// TwinCAT 3 PLC project PLC
// ProgramVersion: 3.1.4026.19
// libraries:
//   Tc2_Standard, * (Beckhoff Automation GmbH)
//   Tc2_System, * (Beckhoff Automation GmbH)
//   Tc2_Utilities, * (Beckhoff Automation GmbH)
//   Tc3_IotBase, * (Beckhoff Automation GmbH)
//   Tc3_IotCommunicator, * (Beckhoff Automation GmbH)
// project tree:
//   DUTs/10-IoT/ ST_IoT_Communicator.TcDUT
//   GVLs/01-System/ GVL_ADS.TcGVL, GVL_NovRam.TcGVL, GVL_System.TcGVL
//   GVLs/02-Knoppen/ GVL_Deurcontacten.TcGVL, GVL_Drukknoppen.TcGVL
//   GVLs/03-Verlichting/ GVL_Dimmers.TcGVL, GVL_Relais.TcGVL
//   GVLs/04-Boiler/ GVL_Boiler.TcGVL
//   GVLs/05-Temperaturen/ GVL_Temperaturen.TcGVL
//   GVLs/06-Screens/ GVL_Screens.TcGVL
//   GVLs/07-Draaipoort/ GVL_Draaipoort.TcGVL
//   GVLs/08-Energiemetingen/ GVL_Energiemetingen.TcGVL
//   GVLs/09-Ventilatie/ GVL_Ventilatie.TcGVL
//   GVLs/90-Visualisatie/ GVL_Visualisatie.TcGVL
//   / PlcTask.TcTTO
//   POUs/00-MAIN/ MAIN.TcPOU
//   POUs/01-System/ P_SunriseSunset.TcPOU, P_WinTime.TcPOU
//   POUs/02-Knoppen/ P_Doors.TcPOU, P_Drukknoppen.TcPOU
//   POUs/03-Verlichting/ P_LightsBerging.TcPOU, P_LightsBoven.TcPOU, P_LightsBuiten.TcPOU, P_LightsHal.TcPOU, P_LightsKeukenLiving.TcPOU, P_LightsLeefruimte.TcPOU
//   POUs/04-Boiler/ P_Boiler.TcPOU
//   POUs/05-Temperaturen/ P_Temperatures.TcPOU
//   POUs/06-Screens/ P_Screens.TcPOU
//   POUs/07-Draaipoort/ P_Draaipoort.TcPOU
//   POUs/08-Energiemetingen/ P_Kwartierpiek.TcPOU, P_Watermeting.TcPOU
//   POUs/09-Ventilatie/ P_Ventilatie.TcPOU
//   POUs/10-IoT/ P_IoT_Communicator.TcPOU, P_Sonos.TcPOU (not stored)
//   POUs/99-FB%27s/ FB_Dimmer.TcPOU (not stored), FB_LongMultipleClick.TcPOU (not stored), FB_OnOffLight.TcPOU (not stored), FB_Screens.TcPOU (not stored)
// real-time tasks:
//   TASK PlcTask: cycle T#10ms, priority 20, ADS port 350
// I/O:
//   DEVICE Device 1 (NOV-DP-RAM)
//     Box 2 (Retain Handler)
//   DEVICE Device 2 (Onboard I/O Device), AmsNetId 5.170.212.74.3.1
//     Term 1 (CX7028) [CX7028-0000-0121]
//       modules: Module 1 (DIO_2x), Module 2 (Empty Module), Module 3 (DIO_2x), Module 4 (Empty Module), Module 5 (DI_2x), Module 6 (Empty Module), Module 7 (DI_2x), Module 8 (Empty Module)
//   DEVICE Device 3 (EtherCAT), AmsNetId 192.168.0.199.4.1
//     Term 1 (EK1200) [EK1200-7000 EtherCAT Power supply (1,5A E-Bus)]
//       DK01-02-03-04 (EL1809) [EL1809 16Ch. Dig. Input 24V, 3ms]
//       DK04-05-06-07 (EL1809) [EL1809 16Ch. Dig. Input 24V, 3ms]
//       DK08-11-12 (EL1809) [EL1809 16Ch. Dig. Input 24V, 3ms]
//       DK13-14-15-16 (EL1809) [EL1809 16Ch. Dig. Input 24V, 3ms]
//       DK09-10 (EL1809) [EL1809 16Ch. Dig. Input 24V, 3ms]
//       Sensoren (EL1008) [EL1008 8Ch. Dig. Input 24V, 3ms]
//       Lights J-K (EL2809) [EL2809 16Ch. Dig. Output 24V, 0.5A]
//       Lights X-Y (EL2809) [EL2809 16Ch. Dig. Output 24V, 0.5A]
//       Boiler en poort (EL2809) [EL2809 16Ch. Dig. Output 24V, 0.5A]
//       Temperaturen (EL3208) [EL3208 8Ch. Ana. Input PT100 (RTD)]
//       Ventilatie en Dimmers1 (EL4004) [EL4004 4Ch. Ana. Output 0-10V, 12bit]
//       Term 15 (EL6851) [EL6851 DMX Master]
//       Term 16 (EL3403) [EL3403 3Ch. Power Measuring]
//       Term 17 (EK1122) [EK1122 2 port EtherCAT junction]
//         Kast Tuinhuis (EK1828) [EK1828 EtherCAT IO-Coupler  (1A E-Bus, 4 Ch. Dig. In, 3ms, 8 Ch. Dig. Out 24V, 0,5A)]
//         Kast Tuinhuis achteraan (EK1828) [EK1828 EtherCAT IO-Coupler  (1A E-Bus, 4 Ch. Dig. In, 3ms, 8 Ch. Dig. Out 24V, 0,5A)]
//         Kast Verdieping (EK1100) [EK1100 EtherCAT Coupler (2A E-Bus)]
//           DK17-18-19 (EL1809) [EL1809 16Ch. Dig. Input 24V, 3ms]
//           DK20-21-22 (EL1809) [EL1809 16Ch. Dig. Input 24V, 3ms]
//           Term 23 (EL1809) [EL1809 16Ch. Dig. Input 24V, 3ms]
//           Screens en Lights-BD (EL2809) [EL2809 16Ch. Dig. Output 24V, 0.5A]
//           Rolluiken (EL2008) [EL2008 8Ch. Dig. Output 24V, 0.5A]
//           Dimmers2 (EL4008) [EL4008 8Ch. Ana. Output 0-10V, 12bit]
//           Term 27 (EL3064) [EL3064 4Ch. Ana. Input 0-10V]
//           Term 26 (EL9011) [EL9011 End Terminal]
// variable links:
//   (this object) <-> Device 1 (NOV-DP-RAM)/Box 2 (Retain Handler)
//     PlcTask Retains/GVL_NovRam.bNovRamBoiler <-> Retains/GVL_NovRam.bNovRamBoiler_[851]
//     PlcTask Retains/GVL_NovRam.bNovRamLight_BD{2..8} <-> Retains/GVL_NovRam.bNovRamLight_BD{2..8}_[851]  (7 links)
//     PlcTask Retains/GVL_NovRam.bNovRamLight_I{1..8} <-> Retains/GVL_NovRam.bNovRamLight_I{1..8}_[851]  (8 links)
//     PlcTask Retains/GVL_NovRam.bNovRamLight_J{3..6} <-> Retains/GVL_NovRam.bNovRamLight_J{3..6}_[851]  (4 links)
//     PlcTask Retains/GVL_NovRam.bNovRamLight_W{1..8} <-> Retains/GVL_NovRam.bNovRamLight_W{1..8}_[851]  (8 links)
//     PlcTask Retains/GVL_NovRam.bNovRamLight_Y{1..7} <-> Retains/GVL_NovRam.bNovRamLight_Y{1..7}_[851]  (7 links)
//     PlcTask Retains/GVL_NovRam.bNovRamLight_Z{1..4} <-> Retains/GVL_NovRam.bNovRamLight_Z{1..4}_[851]  (4 links)
//     PlcTask Retains/GVL_NovRam.bNovRamLight_ZZ{1..6} <-> Retains/GVL_NovRam.bNovRamLight_ZZ{1..6}_[851]  (6 links)
//     PlcTask Retains/GVL_NovRam.diWaterteller <-> Retains/GVL_NovRam.diWaterteller_[851]
//     PlcTask Retains/GVL_NovRam.diWatertellerGisteren <-> Retains/GVL_NovRam.diWatertellerGisteren_[851]
//     PlcTask Retains/GVL_NovRam.iNovRamVentilatie <-> Retains/GVL_NovRam.iNovRamVentilatie_[851]
//     PlcTask Retains/GVL_NovRam.nDimmValue_BD1 <-> Retains/GVL_NovRam.nDimmValue_BD1_[851]
//     PlcTask Retains/GVL_NovRam.nDimmValue_I2 <-> Retains/GVL_NovRam.nDimmValue_I2_[851]
//     PlcTask Retains/GVL_NovRam.nDimmValue_J1 <-> Retains/GVL_NovRam.nDimmValue_J1_[851]
//     PlcTask Retains/GVL_NovRam.nDimmValue_J2 <-> Retains/GVL_NovRam.nDimmValue_J2_[851]
//   (this object) <-> Device 3 (EtherCAT)/Term 1 (EK1200)/Boiler en poort (EL2809)
//     PlcTask Outputs/GVL_Boiler.bRelaisBoiler <-> Channel 1/GVL_Boiler.bRelaisBoiler
//     PlcTask Outputs/GVL_Draaipoort.bDraaipoortVoetgangerOpenDicht <-> Channel 3/GVL_Draaipoort.bDraaipoortVoetgangerOpenDicht
//     PlcTask Outputs/GVL_Draaipoort.bDraaipoortVolledigOpenDicht <-> Channel 2/GVL_Draaipoort.bDraaipoortVolledigOpenDicht
//   (this object) <-> Device 3 (EtherCAT)/Term 1 (EK1200)/DK01-02-03-04 (EL1809)
//     PlcTask Inputs/GVL_Drukknoppen.bDK01x1 <-> Channel 1/GVL_Drukknoppen.bDK01x1
//     PlcTask Inputs/GVL_Drukknoppen.bDK01x2 <-> Channel 2/GVL_Drukknoppen.bDK01x2
//     PlcTask Inputs/GVL_Drukknoppen.bDK01x3 <-> Channel 3/GVL_Drukknoppen.bDK01x3
//     PlcTask Inputs/GVL_Drukknoppen.bDK01x4 <-> Channel 4/GVL_Drukknoppen.bDK01x4
//     PlcTask Inputs/GVL_Drukknoppen.bDK01x5 <-> Channel 5/GVL_Drukknoppen.bDK01x5
//     PlcTask Inputs/GVL_Drukknoppen.bDK01x6 <-> Channel 6/GVL_Drukknoppen.bDK01x6
//     PlcTask Inputs/GVL_Drukknoppen.bDK02x1 <-> Channel 7/GVL_Drukknoppen.bDK02x1
//     PlcTask Inputs/GVL_Drukknoppen.bDK03x1 <-> Channel 9/GVL_Drukknoppen.bDK03x1
//     PlcTask Inputs/GVL_Drukknoppen.bDK03x2 <-> Channel 10/GVL_Drukknoppen.bDK03x2
//     PlcTask Inputs/GVL_Drukknoppen.bDK03x3 <-> Channel 11/GVL_Drukknoppen.bDK03x3
//     PlcTask Inputs/GVL_Drukknoppen.bDK03x4 <-> Channel 12/GVL_Drukknoppen.bDK03x4
//     PlcTask Inputs/GVL_Drukknoppen.bDK04x1 <-> Channel 13/GVL_Drukknoppen.bDK04x1
//     PlcTask Inputs/GVL_Drukknoppen.bDK04x2 <-> Channel 14/GVL_Drukknoppen.bDK04x2
//     PlcTask Inputs/GVL_Drukknoppen.bDK04x3 <-> Channel 15/GVL_Drukknoppen.bDK04x3
//     PlcTask Inputs/GVL_Drukknoppen.bDK04x4 <-> Channel 16/GVL_Drukknoppen.bDK04x4
//   (this object) <-> Device 3 (EtherCAT)/Term 1 (EK1200)/DK04-05-06-07 (EL1809)
//     PlcTask Inputs/GVL_Drukknoppen.bDK04x5 <-> Channel 1/GVL_Drukknoppen.bDK04x5
//     PlcTask Inputs/GVL_Drukknoppen.bDK04x6 <-> Channel 2/GVL_Drukknoppen.bDK04x6
//     PlcTask Inputs/GVL_Drukknoppen.bDK05x1 <-> Channel 3/GVL_Drukknoppen.bDK05x1
//     PlcTask Inputs/GVL_Drukknoppen.bDK05x2 <-> Channel 4/GVL_Drukknoppen.bDK05x2
//     PlcTask Inputs/GVL_Drukknoppen.bDK05x3 <-> Channel 5/GVL_Drukknoppen.bDK05x3
//     PlcTask Inputs/GVL_Drukknoppen.bDK05x4 <-> Channel 6/GVL_Drukknoppen.bDK05x4
//     PlcTask Inputs/GVL_Drukknoppen.bDK06x1 <-> Channel 7/GVL_Drukknoppen.bDK06x1
//     PlcTask Inputs/GVL_Drukknoppen.bDK06x2 <-> Channel 8/GVL_Drukknoppen.bDK06x2
//     PlcTask Inputs/GVL_Drukknoppen.bDK06x3 <-> Channel 9/GVL_Drukknoppen.bDK06x3
//     PlcTask Inputs/GVL_Drukknoppen.bDK06x4 <-> Channel 10/GVL_Drukknoppen.bDK06x4
//     PlcTask Inputs/GVL_Drukknoppen.bDK07x1 <-> Channel 11/GVL_Drukknoppen.bDK07x1
//     PlcTask Inputs/GVL_Drukknoppen.bDK07x2 <-> Channel 12/GVL_Drukknoppen.bDK07x2
//     PlcTask Inputs/GVL_Drukknoppen.bDK07x3 <-> Channel 13/GVL_Drukknoppen.bDK07x3
//     PlcTask Inputs/GVL_Drukknoppen.bDK07x4 <-> Channel 14/GVL_Drukknoppen.bDK07x4
//     PlcTask Inputs/GVL_Drukknoppen.bDK07x5 <-> Channel 15/GVL_Drukknoppen.bDK07x5
//     PlcTask Inputs/GVL_Drukknoppen.bDK07x6 <-> Channel 16/GVL_Drukknoppen.bDK07x6
//   (this object) <-> Device 3 (EtherCAT)/Term 1 (EK1200)/DK08-11-12 (EL1809)
//     PlcTask Inputs/GVL_Drukknoppen.bDK08x1 <-> Channel 1/GVL_Drukknoppen.bDK08x1
//     PlcTask Inputs/GVL_Drukknoppen.bDK08x2 <-> Channel 2/GVL_Drukknoppen.bDK08x2
//     PlcTask Inputs/GVL_Drukknoppen.bDK08x3 <-> Channel 3/GVL_Drukknoppen.bDK08x3
//     PlcTask Inputs/GVL_Drukknoppen.bDK08x4 <-> Channel 4/GVL_Drukknoppen.bDK08x4
//     PlcTask Inputs/GVL_Drukknoppen.bDK11x1 <-> Channel 9/GVL_Drukknoppen.bDK11x1
//     PlcTask Inputs/GVL_Drukknoppen.bDK11x2 <-> Channel 10/GVL_Drukknoppen.bDK11x2
//     PlcTask Inputs/GVL_Drukknoppen.bDK11x3 <-> Channel 11/GVL_Drukknoppen.bDK11x3
//     PlcTask Inputs/GVL_Drukknoppen.bDK11x4 <-> Channel 12/GVL_Drukknoppen.bDK11x4
//     PlcTask Inputs/GVL_Drukknoppen.bDK12x1 <-> Channel 13/GVL_Drukknoppen.bDK12x1
//     PlcTask Inputs/GVL_Drukknoppen.bDK12x2 <-> Channel 14/GVL_Drukknoppen.bDK12x2
//     PlcTask Inputs/GVL_Drukknoppen.bDK12x3 <-> Channel 15/GVL_Drukknoppen.bDK12x3
//     PlcTask Inputs/GVL_Drukknoppen.bDK12x4 <-> Channel 16/GVL_Drukknoppen.bDK12x4
//   (this object) <-> Device 3 (EtherCAT)/Term 1 (EK1200)/DK09-10 (EL1809)
//     PlcTask Inputs/GVL_Drukknoppen.bDK09x1 <-> Channel 1/GVL_Drukknoppen.bDK09x1
//     PlcTask Inputs/GVL_Drukknoppen.bDK09x2 <-> Channel 2/GVL_Drukknoppen.bDK09x2
//     PlcTask Inputs/GVL_Drukknoppen.bDK09x3 <-> Channel 3/GVL_Drukknoppen.bDK09x3
//     PlcTask Inputs/GVL_Drukknoppen.bDK09x4 <-> Channel 4/GVL_Drukknoppen.bDK09x4
//     PlcTask Inputs/GVL_Drukknoppen.bDK09x5 <-> Channel 5/GVL_Drukknoppen.bDK09x5
//     PlcTask Inputs/GVL_Drukknoppen.bDK09x6 <-> Channel 6/GVL_Drukknoppen.bDK09x6
//     PlcTask Inputs/GVL_Drukknoppen.bDK10x1 <-> Channel 7/GVL_Drukknoppen.bDK10x1
//     PlcTask Inputs/GVL_Drukknoppen.bDK10x2 <-> Channel 8/GVL_Drukknoppen.bDK10x2
//     PlcTask Inputs/GVL_Drukknoppen.bDK10x3 <-> Channel 9/GVL_Drukknoppen.bDK10x3
//     PlcTask Inputs/GVL_Drukknoppen.bDK10x4 <-> Channel 10/GVL_Drukknoppen.bDK10x4
//     PlcTask Inputs/GVL_Drukknoppen.bDK10x5 <-> Channel 11/GVL_Drukknoppen.bDK10x5
//     PlcTask Inputs/GVL_Drukknoppen.bDK10x6 <-> Channel 12/GVL_Drukknoppen.bDK10x6
//   (this object) <-> Device 3 (EtherCAT)/Term 1 (EK1200)/DK13-14-15-16 (EL1809)
//     PlcTask Inputs/GVL_Drukknoppen.bDK13x1 <-> Channel 1/GVL_Drukknoppen.bDK13x1
//     PlcTask Inputs/GVL_Drukknoppen.bDK13x2 <-> Channel 2/GVL_Drukknoppen.bDK13x2
//     PlcTask Inputs/GVL_Drukknoppen.bDK13x3 <-> Channel 3/GVL_Drukknoppen.bDK13x3
//     PlcTask Inputs/GVL_Drukknoppen.bDK13x4 <-> Channel 4/GVL_Drukknoppen.bDK13x4
//     PlcTask Inputs/GVL_Drukknoppen.bDK14x1 <-> Channel 5/GVL_Drukknoppen.bDK14x1
//     PlcTask Inputs/GVL_Drukknoppen.bDK14x2 <-> Channel 6/GVL_Drukknoppen.bDK14x2
//     PlcTask Inputs/GVL_Drukknoppen.bDK14x3 <-> Channel 7/GVL_Drukknoppen.bDK14x3
//     PlcTask Inputs/GVL_Drukknoppen.bDK14x4 <-> Channel 8/GVL_Drukknoppen.bDK14x4
//     PlcTask Inputs/GVL_Drukknoppen.bDK15x1 <-> Channel 9/GVL_Drukknoppen.bDK15x1
//     PlcTask Inputs/GVL_Drukknoppen.bDK15x2 <-> Channel 10/GVL_Drukknoppen.bDK15x2
//     PlcTask Inputs/GVL_Drukknoppen.bDK15x3 <-> Channel 11/GVL_Drukknoppen.bDK15x3
//     PlcTask Inputs/GVL_Drukknoppen.bDK15x4 <-> Channel 12/GVL_Drukknoppen.bDK15x4
//     PlcTask Inputs/GVL_Drukknoppen.bDK16x1 <-> Channel 13/GVL_Drukknoppen.bDK16x1
//     PlcTask Inputs/GVL_Drukknoppen.bDK16x2 <-> Channel 14/GVL_Drukknoppen.bDK16x2
//     PlcTask Inputs/GVL_Drukknoppen.bDK16x3 <-> Channel 15/GVL_Drukknoppen.bDK16x3
//     PlcTask Inputs/GVL_Drukknoppen.bDK16x4 <-> Channel 16/GVL_Drukknoppen.bDK16x4
//   (this object) <-> Device 3 (EtherCAT)/Term 1 (EK1200)/Lights J-K (EL2809)
//     PlcTask Outputs/GVL_Drukknoppen.bMeldingDK02x1 <-> Channel 15/GVL_Drukknoppen.bMeldingDK02x1
//     PlcTask Outputs/GVL_Drukknoppen.bMeldingDK11x3 <-> Channel 16/GVL_Drukknoppen.bMeldingDK11x3
//     PlcTask Outputs/GVL_Relais.bRelaisLight_I{1..8} <-> Channel {1..8}/GVL_Relais.bRelaisLight_I{1..8}  (8 links)
//     PlcTask Outputs/GVL_Relais.bRelaisLight_J1 <-> Channel 9/GVL_Relais.bRelaisLight_J1
//     PlcTask Outputs/GVL_Relais.bRelaisLight_J3 <-> Channel 11/GVL_Relais.bRelaisLight_J3
//     PlcTask Outputs/GVL_Relais.bRelaisLight_J4 <-> Channel 12/GVL_Relais.bRelaisLight_J4
//     PlcTask Outputs/GVL_Relais.bRelaisLight_J5 <-> Channel 13/GVL_Relais.bRelaisLight_J5
//     PlcTask Outputs/GVL_Relais.bRelaisLight_J6 <-> Channel 14/GVL_Relais.bRelaisLight_J6
//   (this object) <-> Device 3 (EtherCAT)/Term 1 (EK1200)/Lights X-Y (EL2809)
//     PlcTask Outputs/GVL_Drukknoppen.bMeldingDK11x4 <-> Channel 16/GVL_Drukknoppen.bMeldingDK11x4
//     PlcTask Outputs/GVL_Relais.bRelaisLight_W{1..8} <-> Channel {1..8}/GVL_Relais.bRelaisLight_W{1..8}  (8 links)
//     PlcTask Outputs/GVL_Relais.bRelaisLight_Y{1..7} <-> Channel {9..15}/GVL_Relais.bRelaisLight_Y{1..7}  (7 links)
//   (this object) <-> Device 3 (EtherCAT)/Term 1 (EK1200)/Sensoren (EL1008)
//     PlcTask Inputs/GVL_Deurcontacten.bContactSchuifdeur <-> Channel 3/GVL_Deurcontacten.bContactSchuifdeur
//     PlcTask Inputs/GVL_Deurcontacten.bContactSchuifdeurLeefruimte <-> Channel 4/GVL_Deurcontacten.bContactSchuifdeurLeefruimte
//     PlcTask Inputs/GVL_Deurcontacten.bContactVoordeur <-> Channel 1/GVL_Deurcontacten.bContactVoordeur
//     PlcTask Inputs/GVL_Deurcontacten.bContactZijdeur <-> Channel 2/GVL_Deurcontacten.bContactZijdeur
//     PlcTask Inputs/GVL_Energiemetingen.bWaterSensor <-> Channel 7/GVL_Energiemetingen.bWaterSensor
//   (this object) <-> Device 3 (EtherCAT)/Term 1 (EK1200)/Temperaturen (EL3208)
//     PlcTask Inputs/GVL_Temperaturen.iTemp{1..8} <-> RTD Inputs Channel {1..8}/GVL_Temperaturen.iTemp{1..8}  (8 links)
//   (this object) <-> Device 3 (EtherCAT)/Term 1 (EK1200)/Term 17 (EK1122)/Kast Tuinhuis (EK1828)
//     PlcTask Inputs/GVL_Drukknoppen.bDK30x1 <-> Channel 1/GVL_Drukknoppen.bDK30x1
//     PlcTask Inputs/GVL_Drukknoppen.bDK30x2 <-> Channel 2/GVL_Drukknoppen.bDK30x2
//     PlcTask Outputs/GVL_Relais.bRelaisLight_Z{1..4} <-> Channel {5..8}/GVL_Relais.bRelaisLight_Z{1..4}  (4 links)
//   (this object) <-> Device 3 (EtherCAT)/Term 1 (EK1200)/Term 17 (EK1122)/Kast Tuinhuis achteraan (EK1828)
//     PlcTask Inputs/GVL_Drukknoppen.bDK40x{1..4} <-> Channel {1..4}/GVL_Drukknoppen.bDK40x{1..4}  (4 links)
//     PlcTask Outputs/GVL_Relais.bRelaisLight_ZZ{1..6} <-> Channel {5..10}/GVL_Relais.bRelaisLight_ZZ{1..6}  (6 links)
//   (this object) <-> Device 3 (EtherCAT)/Term 1 (EK1200)/Term 17 (EK1122)/Kast Verdieping (EK1100)/DK17-18-19 (EL1809)
//     PlcTask Inputs/GVL_Drukknoppen.bDK17x1 <-> Channel 1/GVL_Drukknoppen.bDK17x1
//     PlcTask Inputs/GVL_Drukknoppen.bDK17x2 <-> Channel 2/GVL_Drukknoppen.bDK17x2
//     PlcTask Inputs/GVL_Drukknoppen.bDK17x3 <-> Channel 3/GVL_Drukknoppen.bDK17x3
//     PlcTask Inputs/GVL_Drukknoppen.bDK17x4 <-> Channel 4/GVL_Drukknoppen.bDK17x4
//     PlcTask Inputs/GVL_Drukknoppen.bDK17x5 <-> Channel 5/GVL_Drukknoppen.bDK17x5
//     PlcTask Inputs/GVL_Drukknoppen.bDK17x6 <-> Channel 6/GVL_Drukknoppen.bDK17x6
//     PlcTask Inputs/GVL_Drukknoppen.bDK18x1 <-> Channel 7/GVL_Drukknoppen.bDK18x1
//     PlcTask Inputs/GVL_Drukknoppen.bDK18x2 <-> Channel 8/GVL_Drukknoppen.bDK18x2
//     PlcTask Inputs/GVL_Drukknoppen.bDK18x3 <-> Channel 9/GVL_Drukknoppen.bDK18x3
//     PlcTask Inputs/GVL_Drukknoppen.bDK18x4 <-> Channel 10/GVL_Drukknoppen.bDK18x4
//     PlcTask Inputs/GVL_Drukknoppen.bDK19x1 <-> Channel 11/GVL_Drukknoppen.bDK19x1
//     PlcTask Inputs/GVL_Drukknoppen.bDK19x2 <-> Channel 12/GVL_Drukknoppen.bDK19x2
//     PlcTask Inputs/GVL_Drukknoppen.bDK19x3 <-> Channel 13/GVL_Drukknoppen.bDK19x3
//     PlcTask Inputs/GVL_Drukknoppen.bDK19x4 <-> Channel 14/GVL_Drukknoppen.bDK19x4
//     PlcTask Inputs/GVL_Drukknoppen.bDK19x5 <-> Channel 15/GVL_Drukknoppen.bDK19x5
//     PlcTask Inputs/GVL_Drukknoppen.bDK19x6 <-> Channel 16/GVL_Drukknoppen.bDK19x6
//   (this object) <-> Device 3 (EtherCAT)/Term 1 (EK1200)/Term 17 (EK1122)/Kast Verdieping (EK1100)/DK20-21-22 (EL1809)
//     PlcTask Inputs/GVL_Drukknoppen.bDK20x1 <-> Channel 1/GVL_Drukknoppen.bDK20x1
//     PlcTask Inputs/GVL_Drukknoppen.bDK20x2 <-> Channel 2/GVL_Drukknoppen.bDK20x2
//     PlcTask Inputs/GVL_Drukknoppen.bDK20x3 <-> Channel 3/GVL_Drukknoppen.bDK20x3
//     PlcTask Inputs/GVL_Drukknoppen.bDK20x4 <-> Channel 4/GVL_Drukknoppen.bDK20x4
//     PlcTask Inputs/GVL_Drukknoppen.bDK21x1 <-> Channel 5/GVL_Drukknoppen.bDK21x1
//     PlcTask Inputs/GVL_Drukknoppen.bDK21x2 <-> Channel 6/GVL_Drukknoppen.bDK21x2
//     PlcTask Inputs/GVL_Drukknoppen.bDK21x3 <-> Channel 7/GVL_Drukknoppen.bDK21x3
//     PlcTask Inputs/GVL_Drukknoppen.bDK21x4 <-> Channel 8/GVL_Drukknoppen.bDK21x4
//     PlcTask Inputs/GVL_Drukknoppen.bDK22x1 <-> Channel 9/GVL_Drukknoppen.bDK22x1
//     PlcTask Inputs/GVL_Drukknoppen.bDK22x2 <-> Channel 10/GVL_Drukknoppen.bDK22x2
//     PlcTask Inputs/GVL_Drukknoppen.bDK22x3 <-> Channel 11/GVL_Drukknoppen.bDK22x3
//     PlcTask Inputs/GVL_Drukknoppen.bDK22x4 <-> Channel 12/GVL_Drukknoppen.bDK22x4
//   (this object) <-> Device 3 (EtherCAT)/Term 1 (EK1200)/Term 17 (EK1122)/Kast Verdieping (EK1100)/Dimmers2 (EL4008)
//     PlcTask Outputs/GVL_Dimmers.DimLight_BD1 <-> AO Outputs Channel 1/GVL_Dimmers.DimLight_BD1
//   (this object) <-> Device 3 (EtherCAT)/Term 1 (EK1200)/Term 17 (EK1122)/Kast Verdieping (EK1100)/Rolluiken (EL2008)
//     PlcTask Outputs/GVL_Screens.bMotorRolluik2Omhoog <-> Channel 1/GVL_Screens.bMotorRolluik2Omhoog
//     PlcTask Outputs/GVL_Screens.bMotorRolluik3Omhoog <-> Channel 3/GVL_Screens.bMotorRolluik3Omhoog
//     PlcTask Outputs/GVL_Screens.bMotorRolluik2Omlaag <-> Channel 2/GVL_Screens.bMotorRolluik2Omlaag
//     PlcTask Outputs/GVL_Screens.bMotorRolluik3Omlaag <-> Channel 4/GVL_Screens.bMotorRolluik3Omlaag
//   (this object) <-> Device 3 (EtherCAT)/Term 1 (EK1200)/Term 17 (EK1122)/Kast Verdieping (EK1100)/Screens en Lights-BD (EL2809)
//     PlcTask Outputs/GVL_Relais.bRelaisLight_BD2 <-> Channel 11/GVL_Relais.bRelaisLight_BD2
//     PlcTask Outputs/GVL_Relais.bRelaisLight_BD3 <-> Channel 12/GVL_Relais.bRelaisLight_BD3
//     PlcTask Outputs/GVL_Relais.bRelaisLight_BD4 <-> Channel 13/GVL_Relais.bRelaisLight_BD4
//     PlcTask Outputs/GVL_Relais.bRelaisLight_BD5 <-> Channel 14/GVL_Relais.bRelaisLight_BD5
//     PlcTask Outputs/GVL_Relais.bRelaisLight_BD6 <-> Channel 15/GVL_Relais.bRelaisLight_BD6
//     PlcTask Outputs/GVL_Relais.bRelaisLight_BD8 <-> Channel 16/GVL_Relais.bRelaisLight_BD8
//     PlcTask Outputs/GVL_Screens.bMotorRolluik1Omhoog <-> Channel 9/GVL_Screens.bMotorRolluik1Omhoog
//     PlcTask Outputs/GVL_Screens.bMotorRolluik1Omlaag <-> Channel 10/GVL_Screens.bMotorRolluik1Omlaag
//     PlcTask Outputs/GVL_Screens.bMotorScreen{1..4}Omhoog <-> Channel {1..7 step 2}/GVL_Screens.bMotorScreen{1..4}Omhoog  (4 links)
//     PlcTask Outputs/GVL_Screens.bMotorScreen{1..4}Omlaag <-> Channel {2..8 step 2}/GVL_Screens.bMotorScreen{1..4}Omlaag  (4 links)
//   (this object) <-> Device 3 (EtherCAT)/Term 1 (EK1200)/Ventilatie en Dimmers1 (EL4004)
//     PlcTask Outputs/GVL_Dimmers.DimLight_I2 <-> AO Outputs Channel 2/GVL_Dimmers.DimLight_I2
//     PlcTask Outputs/GVL_Dimmers.DimLight_J1 <-> AO Outputs Channel 4/GVL_Dimmers.DimLight_J1
//     PlcTask Outputs/GVL_Dimmers.DimLight_J2 <-> AO Outputs Channel 3/GVL_Dimmers.DimLight_J2
//     PlcTask Outputs/GVL_Ventilatie.iVentilatie <-> AO Outputs Channel 1/GVL_Ventilatie.iVentilatie

CONFIGURATION PLC
    RESOURCE PLC ON TwinCAT3
        TASK PlcTask(INTERVAL := T#10ms, PRIORITY := 20);
        PROGRAM MAIN WITH PlcTask : MAIN;
    END_RESOURCE
END_CONFIGURATION

// ---- DUTs/10-IoT/ST_IoT_Communicator.TcDUT
TYPE ST_IoT_Communicator :
STRUCT
	{attribute 'iot.DisplayName' := 'Actief Vermogen'}
	{attribute 'iot.Unit' := 'W'}
	{attribute 'iot.ReadOnly' := 'TRUE'}
	{attribute 'iot.DecimalPrecision' := '1'}
	rActiefVermogen	: REAL;
	
	{attribute 'iot.DisplayName' := 'Keuken'}
    bLampKeuken : BOOL;
END_STRUCT
END_TYPE

// ---- GVLs/01-System/GVL_ADS.TcGVL
//{attribute 'qualified_only'}
VAR_GLOBAL
	bAdsSunIsDown					: BOOL;
                            		
	bAdsAllScreensUp				: BOOL;
	bAdsAllScreensDn				: BOOL;
	bAdsScreen2Up					: BOOL;
	bAdsScreen2Dn					: BOOL;
	bAdsScreen13Up					: BOOL;
	bAdsScreen13Dn					: BOOL;
	bAdsScreen4Up					: BOOL;
	bAdsScreen4Dn					: BOOL;
                            		
	bAdsLichtKeukenCentraal			: BOOL;
	bAdsLichtKeukenSpotsDampkap		: BOOL;
	bAdsLichtLivingStepUp			: BOOL;
	bAdsLichtLivingStepDown			: BOOL;

	bAdsPoortOpenDicht				: BOOL;
	bAdsPoortVoetganger				: BOOL;

	bAdsBoilerOnOff					: BOOL;
	bAdsBoilerState					: BOOL;

	bAdsSonosBadkamerPause			: BOOL;
	bAdsSonosBadkamerPlaylist1		: BOOL;
	bAdsSonosBadkamerPlaylist2	 	: BOOL;
END_VAR

// ---- GVLs/01-System/GVL_NovRam.TcGVL
//{attribute 'qualified_only'}
VAR_GLOBAL RETAIN
	(**********************************************************************)
	(*********************** IMPULSRELAIS **************************)
	(**********************************************************************)
	bNovRamLight_I1 	: BOOL;
	bNovRamLight_I2		: BOOL;
	bNovRamLight_I3 	: BOOL;
	bNovRamLight_I4 	: BOOL;
	bNovRamLight_I5 	: BOOL;
	bNovRamLight_I6 	: BOOL;
	bNovRamLight_I7 	: BOOL;
	bNovRamLight_I8 	: BOOL;

	(*bNovRamLight_J1 	: BOOL;*)
	(*bNovRamLight_J2 	: BOOL;*)
	bNovRamLight_J3 	: BOOL;
	bNovRamLight_J4 	: BOOL;
	bNovRamLight_J5 	: BOOL;
	bNovRamLight_J6 	: BOOL;

	bNovRamLight_W1  	: BOOL;
	bNovRamLight_W2  	: BOOL;
	bNovRamLight_W3  	: BOOL;
	bNovRamLight_W4  	: BOOL;
	bNovRamLight_W5  	: BOOL;
	bNovRamLight_W6  	: BOOL;
	bNovRamLight_W7  	: BOOL;
	bNovRamLight_W8  	: BOOL;

	bNovRamLight_Y1 	: BOOL;
	bNovRamLight_Y2 	: BOOL;
	bNovRamLight_Y3 	: BOOL;
	bNovRamLight_Y4 	: BOOL;
	bNovRamLight_Y5 	: BOOL;
	bNovRamLight_Y6 	: BOOL;
	bNovRamLight_Y7 	: BOOL;

	bNovRamLight_Z1 	: BOOL;
	bNovRamLight_Z2 	: BOOL;
	bNovRamLight_Z3 	: BOOL;
	bNovRamLight_Z4 	: BOOL;

	bNovRamLight_BD2 	: BOOL;
	bNovRamLight_BD3 	: BOOL;
	bNovRamLight_BD4 	: BOOL;
	bNovRamLight_BD5 	: BOOL;
	bNovRamLight_BD6 	: BOOL;
	bNovRamLight_BD7 	: BOOL;
	bNovRamLight_BD8 	: BOOL;

	bNovRamLight_ZZ1 	: BOOL;
	bNovRamLight_ZZ2 	: BOOL;
	bNovRamLight_ZZ3 	: BOOL;
	bNovRamLight_ZZ4 	: BOOL;
	bNovRamLight_ZZ5 	: BOOL;
	bNovRamLight_ZZ6 	: BOOL;

	(**********************************************************************)
	(*********************** DIMMERS *********************************)
	(**********************************************************************)
	nDimmValue_I2		: UINT;
	nDimmValue_BD1		: UINT;
	nDimmValue_J2		: UINT;
	nDimmValue_J1		: UINT;




	(**********************************************************************)
	(*********************** VENTILATIE ******************************)
	(**********************************************************************)
	iNovRamVentilatie 	: INT;



	(**********************************************************************)
	(*********************** BOILER ************************************)
	(**********************************************************************)
	bNovRamBoiler 		: BOOL;



	(**********************************************************************)
	(*********************** ENERGIEMETING ***********************)
	(**********************************************************************)
	diWaterteller			: DINT;
	diWatertellerGisteren	: DINT;
END_VAR

// ---- GVLs/01-System/GVL_System.TcGVL
//{attribute 'qualified_only'}
VAR_GLOBAL
	(* Windows Time Variables *)
	strWinTime				: TIMESTRUCT;
	todWinTime				: TOD;
	sTime					: STRING;
	sDate					: STRING;
	bValidSystemTime		: BOOL;
	bMiddernacht			: BOOL;

END_VAR

// ---- GVLs/02-Knoppen/GVL_Deurcontacten.TcGVL
//{attribute 'qualified_only'}
VAR_GLOBAL
	bContactVoordeur				AT %I*	: BOOL;
	bContactZijdeur					AT %I*	: BOOL;
	bContactSchuifdeur				AT %I*	: BOOL;
	bContactSchuifdeurLeefruimte	AT %I*	: BOOL;
END_VAR

// ---- GVLs/02-Knoppen/GVL_Drukknoppen.TcGVL
//{attribute 'qualified_only'}
VAR_GLOBAL
	(**********************************************************************)
	(*********************** GELIJKVLOERS **************************)
	(**********************************************************************)
	(* Zijdeur *)
	bDK01x1	AT 	%I*	: BOOL;
	bDK01x2	AT 	%I*	: BOOL;
	bDK01x3	AT 	%I*	: BOOL;
	bDK01x4	AT 	%I*	: BOOL;
	bDK01x5	AT 	%I*	: BOOL;
	bDK01x6	AT 	%I*	: BOOL;

	(* WC beneden *)
	bDK02x1	AT 	%I*	: BOOL;

	(* Berging 1 *)
	bDK03x1	AT 	%I* : BOOL;
	bDK03x2	AT 	%I*	: BOOL;
	bDK03x3	AT 	%I*	: BOOL;
	bDK03x4	AT 	%I*	: BOOL;

	(* Schuifraam keuken *)
	bDK04x1	AT 	%I*	: BOOL;
	bDK04x2	AT 	%I*	: BOOL;
	bDK04x3	AT 	%I*	: BOOL;
	bDK04x4	AT 	%I*	: BOOL;
	bDK04x5	AT 	%I*	: BOOL;
	bDK04x6	AT 	%I*	: BOOL;

	(* Kookvuur *)
	bDK05x1	AT 	%I*	: BOOL;
	bDK05x2	AT 	%I*	: BOOL;
	bDK05x3	AT 	%I*	: BOOL;
	bDK05x4	AT 	%I*	: BOOL;

	(* Kookeiland *)
	bDK06x1	AT 	%I*	: BOOL;
	bDK06x2	AT 	%I*	: BOOL;
	bDK06x3	AT 	%I*	: BOOL;
	bDK06x4	AT 	%I*	: BOOL;

	(* Living *)
	bDK07x1	AT 	%I*	: BOOL;
	bDK07x2	AT 	%I*	: BOOL;
	bDK07x3	AT 	%I*	: BOOL;
	bDK07x4	AT 	%I*	: BOOL;
	bDK07x5	AT 	%I*	: BOOL;
	bDK07x6	AT 	%I*	: BOOL;

	(* Voordeur *)
	bDK08x1	AT 	%I*	: BOOL;
	bDK08x2	AT 	%I*	: BOOL;
	bDK08x3	AT 	%I*	: BOOL;
	bDK08x4	AT 	%I*	: BOOL;

	(* Leefruimte tegen keuken *)
	bDK09x1	AT 	%I*	: BOOL;
	bDK09x2	AT 	%I*	: BOOL;
	bDK09x3	AT 	%I*	: BOOL;
	bDK09x4	AT 	%I*	: BOOL;
	bDK09x5	AT 	%I*	: BOOL;
	bDK09x6	AT 	%I*	: BOOL;

	(* Leefruimte tegen buitenmuur *)
	bDK10x1	AT 	%I*	: BOOL;
	bDK10x2	AT 	%I*	: BOOL;
	bDK10x3	AT 	%I*	: BOOL;
	bDK10x4	AT 	%I*	: BOOL;
	bDK10x5	AT 	%I*	: BOOL;
	bDK10x6	AT 	%I*	: BOOL;


	(**********************************************************************)
	(*********************** VERDIEPING *****************************)
	(**********************************************************************)
	(* Traphal *)
	bDK11x1	AT 	%I*	: BOOL;
	bDK11x2	AT 	%I*	: BOOL;
	bDK11x3	AT 	%I*	: BOOL;
	bDK11x4	AT 	%I*	: BOOL;

	(* Badkamer 1 *)
	bDK12x1	AT 	%I*	: BOOL;
	bDK12x2	AT 	%I*	: BOOL;
	bDK12x3	AT 	%I*	: BOOL;
	bDK12x4	AT 	%I*	: BOOL;

	(* Berging 2 deur*)
	bDK13x1	AT 	%I*	: BOOL;
	bDK13x2	AT 	%I*	: BOOL;
	bDK13x3	AT 	%I*	: BOOL;
	bDK13x4	AT 	%I*	: BOOL;

	(* Berging 2 wand *)
	bDK14x1	AT 	%I*	: BOOL;
	bDK14x2	AT 	%I*	: BOOL;
	bDK14x3	AT 	%I*	: BOOL;
	bDK14x4	AT 	%I*	: BOOL;

	(* Slaapkamer 2 deur *)
	bDK15x1	AT 	%I*	: BOOL;
	bDK15x2	AT 	%I*	: BOOL;
	bDK15x3	AT 	%I*	: BOOL;
	bDK15x4	AT 	%I*	: BOOL;

	(* Slaapkamer 3 deur *)
	bDK16x1	AT 	%I*	: BOOL;
	bDK16x2	AT 	%I*	: BOOL;
	bDK16x3	AT 	%I*	: BOOL;
	bDK16x4	AT 	%I*	: BOOL;

	(* Slaapkamer 1 deur *)
	bDK17x1	AT 	%I*	: BOOL;
	bDK17x2	AT 	%I*	: BOOL;
	bDK17x3	AT 	%I*	: BOOL;
	bDK17x4	AT 	%I*	: BOOL;
	bDK17x5	AT 	%I*	: BOOL;
	bDK17x6	AT 	%I*	: BOOL;

	(* Slaapkamer 1 wand *)
	bDK18x1	AT 	%I*	: BOOL;
	bDK18x2	AT 	%I*	: BOOL;
	bDK18x3	AT 	%I*	: BOOL;
	bDK18x4	AT 	%I*	: BOOL;

	(* Slaapkamer 1 raam *)
	bDK19x1	AT 	%I*	: BOOL;
	bDK19x2	AT 	%I*	: BOOL;
	bDK19x3	AT 	%I*	: BOOL;
	bDK19x4	AT 	%I*	: BOOL;
	bDK19x5	AT 	%I*	: BOOL;
	bDK19x6	AT 	%I*	: BOOL;

	(* Slaapkamer 1 deur badkamer 2 *)
	bDK20x1	AT 	%I*	: BOOL;
	bDK20x2	AT 	%I*	: BOOL;
	bDK20x3	AT 	%I*	: BOOL;
	bDK20x4	AT 	%I*	: BOOL;

	(* Badkamer 2 deur *)
	bDK21x1	AT 	%I*	: BOOL;
	bDK21x2	AT 	%I*	: BOOL;
	bDK21x3	AT 	%I*	: BOOL;
	bDK21x4	AT 	%I*	: BOOL;

	(* Badkamer 2 wand *)
	bDK22x1	AT 	%I*	: BOOL;
	bDK22x2	AT 	%I*	: BOOL;
	bDK22x3	AT 	%I*	: BOOL;
	bDK22x4	AT 	%I*	: BOOL;


	(**********************************************************************)
	(*********************** BUITEN ************************************)
	(**********************************************************************)
	(* Tuinhuis binnen *)
	bDK30x1	AT 	%I*	: BOOL;
	bDK30x2	AT 	%I*	: BOOL;

	(* Tuinhuis achteraan - 4 voudige knop binnen*)
	bDK40x1 AT 	%I*	: BOOL;
	bDK40x2 AT 	%I*	: BOOL;
	bDK40x3 AT 	%I*	: BOOL;
	bDK40x4 AT 	%I*	: BOOL;

	(**********************************************************************)
	(*********************** MELDING DRUKKNOPPEN *************)
	(**********************************************************************)
	bMeldingDK02x1	AT 	%Q*	: BOOL;
	bMeldingDK11x3	AT 	%Q*	: BOOL;
	bMeldingDK11x4	AT 	%Q* : BOOL;


	(* Alles uit *)
	bAllOff			: BOOL;
	bAllOffBeneden	: BOOL;

	(* Multiple click *)
	fbShortLongClick12x3: FB_LongMultipleClick;
	fbShortLongClick21x3: FB_LongMultipleClick;
	fbShortLongClick22x3: FB_LongMultipleClick;
	fbShortLongClick22x4: FB_LongMultipleClick;
	fbShortLongClick30x1: FB_LongMultipleClick;
	fbShortLongClick30x2: FB_LongMultipleClick;
END_VAR

// ---- GVLs/03-Verlichting/GVL_Dimmers.TcGVL
//{attribute 'qualified_only'}
VAR_GLOBAL
	(* Dimmer outputs *)
	DimLight_I2 	AT %Q*: INT;
	DimLight_BD1 	AT %Q*: INT;
	DimLight_J2 	AT %Q*: INT;
	DimLight_J1 	AT %Q*: INT;
	(*DimLight_J3 	AT %Q*: INT;*)

	tDimmerTijd		: TIME := T#5S;

	(* Dimmers *)
	fbDimmer_I2		: FB_Dimmer;
	fbDimmer_J1		: FB_Dimmer;
	fbDimmer_J2		: FB_Dimmer;
	fbDimmer_BD1	: FB_Dimmer;
	(*fbDimmer_J3	: FB_Dimmer2Switch;*)

END_VAR

// ---- GVLs/03-Verlichting/GVL_Relais.TcGVL
//{attribute 'qualified_only'}
VAR_GLOBAL
	(**********************************************************************)
	(*********************** IMPULSRELAIS **************************)
	(**********************************************************************)
	bRelaisLight_I1 AT %Q*	: BOOL;	(* Centraalpunt Hal *)
	bRelaisLight_I2 AT %Q*	: BOOL;	(* Niet gebruikt. Was Centraalpunt Living *)
	bRelaisLight_I3 AT %Q*	: BOOL;	(* Geschakeld stopcontact living *)
	bRelaisLight_I4 AT %Q*	: BOOL;	(* Button+ voeding *)
	bRelaisLight_I5 AT %Q*	: BOOL;	(* Centraalpunt Keuken *)
	bRelaisLight_I6 AT %Q*	: BOOL;	(* Verlichting onder kookeiland *)			(* Niet aangesloten *)
	bRelaisLight_I7 AT %Q*	: BOOL;	(* Spots naast dampkap *)
	bRelaisLight_I8 AT %Q*	: BOOL;	(* Nog verwijderen, niet meer in gebruik. Was verlichting led strip boven keukenkast *)
                          	
	bRelaisLight_J1 AT %Q*	: BOOL;	(* Niet meer in gebruik. Was centraal Slaapkamer 3 *)
	(*bRelaisLight_J2 AT %Q*: BOOL;	(* Niet meer in gebruik. Was centraal Slaapkamer 2 *)*)
	bRelaisLight_J3 AT %Q*	: BOOL;	(* Centraal Slaapkamer 1 boven *)
	bRelaisLight_J4 AT %Q*	: BOOL;	(* 3 spots Slaapkamer 1 boven *)
	bRelaisLight_J5 AT %Q*	: BOOL;	(* 4 spots Plafond traphal *)
	bRelaisLight_J6 AT %Q*	: BOOL;	(* 5 spots muur traphal *)
                          	
	bRelaisLight_W1 AT %Q*	: BOOL;	(* Spot WC beneden *)
	bRelaisLight_W2 AT %Q*	: BOOL;	(* Verlichting boven pompbak berging *)
	bRelaisLight_W3 AT %Q*	: BOOL;	(* Centraalpunt berging *)
	bRelaisLight_W4 AT %Q*	: BOOL;	(* Centraalpunt koele berging *)
	bRelaisLight_W5 AT %Q*	: BOOL;	(* Spot douche *)
	bRelaisLight_W6 AT %Q*	: BOOL;	(* Spot WC badkamer *)
	bRelaisLight_W7 AT %Q*	: BOOL;	(* Centraal badkamer *)
	bRelaisLight_W8 AT %Q*	: BOOL;	(* Centraal technische ruimte boven *)
                          	
	bRelaisLight_Y1 AT %Q*	: BOOL;	(* Leefruimte Spots barkast *)
	bRelaisLight_Y2 AT %Q*	: BOOL;	(* Leefruimte Centraal eettafel *)
	bRelaisLight_Y3 AT %Q*	: BOOL;	(* Leefruimte Spots zithoek *)
	bRelaisLight_Y4 AT %Q*	: BOOL;	(* Muurverlichting carport *)
	bRelaisLight_Y5 AT %Q*	: BOOL;	(* Muurverlichting leefruimte up/down spots *)
	bRelaisLight_Y6 AT %Q*	: BOOL;	(* Robotmaaier stopcontact *)
	bRelaisLight_Y7 AT %Q*	: BOOL;	(* Muurverlichting voorgevel up/down spots *)
                          	
	bRelaisLight_Z1 AT %Q*	: BOOL;	(* TL lampen tuinhuis *)
	bRelaisLight_Z2 AT %Q*	: BOOL;	(* 5 spots zijkant tuinhuis *)
	bRelaisLight_Z3 AT %Q*	: BOOL;	(* Verlichting vuilbakken *)
	bRelaisLight_Z4 AT %Q*	: BOOL;	(* Geschakeld stopcontact tuinhuis *)

	bRelaisLight_BD2 AT %Q*	: BOOL;	(* Spots kleerkast slaapkamer 1 *)
	bRelaisLight_BD3 AT %Q*	: BOOL;	(* Spots dressoir slaapkamer 1 *)
	bRelaisLight_BD4 AT %Q*	: BOOL;	(* Spots bad *)
	bRelaisLight_BD5 AT %Q*	: BOOL;	(* Spots badkamer 2 *)
	bRelaisLight_BD6 AT %Q*	: BOOL;	(* Spots spiegel badkamer 2 *)
	bRelaisLight_BD7 AT %Q*	: BOOL;	(* Leefruimte Centraal zithoek *)
	bRelaisLight_BD8 AT %Q*	: BOOL;	(* 2 Spots buitengevel leefruimte op terras *)
                           	
	bRelaisLight_ZZ1 AT %Q*	: BOOL;	(* Centrale spots tuinhuis achteraan *)
	bRelaisLight_ZZ2 AT %Q*	: BOOL;	(* 2 spots wand tuinhuis achteraan *)
	bRelaisLight_ZZ3 AT %Q*	: BOOL;
	bRelaisLight_ZZ4 AT %Q*	: BOOL;
	bRelaisLight_ZZ5 AT %Q*	: BOOL;
	bRelaisLight_ZZ6 AT %Q*	: BOOL;
END_VAR

// ---- GVLs/04-Boiler/GVL_Boiler.TcGVL
//{attribute 'qualified_only'}
VAR_GLOBAL
	bRelaisBoiler 		AT %Q*	: BOOL;	(* Geschakeld stopcontact *)
END_VAR

// ---- GVLs/05-Temperaturen/GVL_Temperaturen.TcGVL
//{attribute 'qualified_only'}
VAR_GLOBAL
	iTemp1 	AT %I*:	INT;
	iTemp2 	AT %I*:	INT;
	iTemp3 	AT %I*:	INT;
	iTemp4 	AT %I*:	INT;
	iTemp5 	AT %I*:	INT;
	iTemp6 	AT %I*:	INT;
	iTemp7 	AT %I*:	INT;
	iTemp8 	AT %I*:	INT;
END_VAR

// ---- GVLs/06-Screens/GVL_Screens.TcGVL
//{attribute 'qualified_only'}
VAR_GLOBAL
	bMotorScreen1Omhoog		AT %Q*: BOOL;
	bMotorScreen1Omlaag		AT %Q*: BOOL;
	bMotorScreen2Omhoog		AT %Q*: BOOL;
	bMotorScreen2Omlaag		AT %Q*: BOOL;
	bMotorScreen3Omhoog		AT %Q*: BOOL;
	bMotorScreen3Omlaag		AT %Q*: BOOL;
	bMotorScreen4Omhoog		AT %Q*: BOOL;
	bMotorScreen4Omlaag		AT %Q*: BOOL;

	bMotorRolluik1Omhoog	AT %Q*: BOOL;
	bMotorRolluik1Omlaag	AT %Q*: BOOL;
	bMotorRolluik2Omhoog	AT %Q*: BOOL;
	bMotorRolluik2Omlaag	AT %Q*: BOOL;
	bMotorRolluik3Omhoog	AT %Q*: BOOL;
	bMotorRolluik3Omlaag	AT %Q*: BOOL;
END_VAR

// ---- GVLs/07-Draaipoort/GVL_Draaipoort.TcGVL
//{attribute 'qualified_only'}
VAR_GLOBAL
	bDraaipoortVolledigOpenDicht	AT %Q*	: BOOL;
	bDraaipoortVoetgangerOpenDicht	AT %Q*	: BOOL;
END_VAR

// ---- GVLs/08-Energiemetingen/GVL_Energiemetingen.TcGVL
//{attribute 'qualified_only'}
VAR_GLOBAL
	bWaterSensor 			AT %I*	: BOOL;
	diWaterverbruikVandaag			: DINT;
END_VAR

// ---- GVLs/09-Ventilatie/GVL_Ventilatie.TcGVL
//{attribute 'qualified_only'}
VAR_GLOBAL
	iVentilatie		AT %Q*	: INT;
	
	bVentUp					: BOOL;
	bVentDown				: BOOL;
END_VAR

// ---- GVLs/90-Visualisatie/GVL_Visualisatie.TcGVL
//{attribute 'qualified_only'}
VAR_GLOBAL
	(* Virtuele bediening lampen *)
	bVLight_I1:		BOOL;
	bVLight_I2:		BOOL;
	bVLight_I3:		BOOL;
	bVLight_I4:		BOOL;
	bVLight_I5:		BOOL;
	bVLight_I6:		BOOL;
	bVLight_I7:		BOOL;
	bVLight_I8:		BOOL;

	bVLight_J1:		BOOL;
	bVLight_J2:		BOOL;
	bVLight_J3:		BOOL;
	bVLight_J4:		BOOL;
	bVLight_J5:		BOOL;
	bVLight_J6:		BOOL;

	bVLight_W1:		BOOL;
	bVLight_W2:		BOOL;
	bVLight_W3:		BOOL;
	bVLight_W4:		BOOL;
	bVLight_W5:		BOOL;
	bVLight_W6:		BOOL;
	bVLight_W7:		BOOL;
	bVLight_W8:		BOOL;

	bVLight_Y1:		BOOL;
	bVLight_Y2:		BOOL;
	bVLight_Y3:		BOOL;
	bVLight_Y4:		BOOL;
	bVLight_Y5:		BOOL;
	bVLight_Y6:		BOOL;
	bVLight_Y7:		BOOL;

	bVLight_Z1:		BOOL;
	bVLight_Z2:		BOOL;
	bVLight_Z3:		BOOL;
	bVLight_Z4:		BOOL;

	bVLedUp:		BOOL;
	bVLedDn:		BOOL;
	bVLedNext:		BOOL;

	bVLuifelin:		BOOL;
	bVLuifeluit:	BOOL;
END_VAR

// ---- POUs/00-MAIN/MAIN.TcPOU
PROGRAM MAIN
VAR
END_VAR

P_SunriseSunset();
P_WinTime();

P_Doors();
P_Drukknoppen();

P_LightsBerging();
P_LightsBoven();
P_LightsBuiten();
P_LightsHal();
P_LightsKeukenLiving();
P_LightsLeefruimte();

P_Boiler();

P_Temperatures();

P_Screens();

P_Draaipoort();

P_Kwartierpiek();
P_Watermeting();

P_Ventilatie();

P_IoT_Communicator();
P_Sonos();

END_PROGRAM

// ---- POUs/01-System/P_SunriseSunset.TcPOU
PROGRAM P_SunriseSunset
VAR
	bSunsetPulse		: BOOL;
	bSunrisePulse		: BOOL;

	rtSunset			: R_TRIG;
	ftSunset			: F_TRIG;
END_VAR

rtSunset(CLK:=bAdsSunIsDown, Q=>bSunsetPulse);
ftSunset(CLK:=bAdsSunIsDown, Q=>bSunrisePulse);

END_PROGRAM

// ---- POUs/01-System/P_WinTime.TcPOU
PROGRAM P_WinTime
VAR
	GetLocalSystemTime	: FB_LocalSystemTime;
	bEnable				: BOOL := TRUE;
END_VAR

GetLocalSystemTime(
	sNetID:= ,
	bEnable:= bEnable,
	dwCycle:= ,
	dwOpt:= ,
	tTimeout:= ,
	bValid=> bValidSystemTime,
	systemTime=>strWinTime ,
	tzID=> );

todWinTime := LREAL_TO_TOD(strWinTime.wHour*3600000 + strWinTime.wMinute*60000 + strWinTime.wSecond*1000);

sTime := 	CONCAT(	CONCAT(WORD_TO_STRING(strWinTime.wHour),':'),
					CONCAT(
								CONCAT(WORD_TO_STRING(strWinTime.wMinute),':'),
								WORD_TO_STRING(strWinTime.wSecond)
							)
				);

sDate :=	CONCAT(	CONCAT(WORD_TO_STRING(strWinTime.wYear),'-'),
					CONCAT(
								CONCAT(WORD_TO_STRING(strWinTime.wMonth),'-'),
								WORD_TO_STRING(strWinTime.wDay)
							)
				);

bMiddernacht := todWinTime = TOD#00:00:00;

END_PROGRAM

// ---- POUs/02-Knoppen/P_Doors.TcPOU
PROGRAM P_Doors
VAR
	ftContactVoordeur				: F_TRIG;
	ftContactZijdeur				: F_TRIG;
	ftContactSchuifdeur				: F_TRIG;
	ftContactSchuifdeurLeefruimte	: F_TRIG;
END_VAR

ftContactVoordeur(CLK:= bContactVoordeur, Q=> );
ftContactZijdeur(CLK:= bContactZijdeur, Q=> );
ftContactSchuifdeur(CLK:= bContactSchuifdeur, Q=> );
ftContactSchuifdeurLeefruimte(CLK:= bContactSchuifdeurLeefruimte, Q=> );

END_PROGRAM

// ---- POUs/02-Knoppen/P_Drukknoppen.TcPOU
PROGRAM P_Drukknoppen
VAR
END_VAR

fbShortLongClick12x3(bInput:= bDK12x3 );
fbShortLongClick21x3(bInput:= bDK21x3 );
fbShortLongClick22x3(bInput:= bDK22x3 );
fbShortLongClick22x4(bInput:= bDK22x4 );
fbShortLongClick30x1(bInput:= bDK30x1 );
fbShortLongClick30x2(bInput:= bDK30x2 );

END_PROGRAM

// ---- POUs/03-Verlichting/P_LightsBerging.TcPOU
PROGRAM P_LightsBerging
VAR
	bSwitchLight_W1	: BOOL;
	bSwitchLight_W2	: BOOL;
	bSwitchLight_W3	: BOOL;
	bSwitchLight_W4	: BOOL;

	fbOnOffLight_W1	: FB_OnOffLight;
	fbOnOffLight_W2	: FB_OnOffLight;
	fbOnOffLight_W3	: FB_OnOffLight;
	fbOnOffLight_W4	: FB_OnOffLight;
END_VAR


//Berging en Koele berging
bSwitchLight_W1 := bVLight_W1 OR bDK02x1;					//Licht WC
bSwitchLight_W2 := bVLight_W2 OR bDK03x3;					//Licht Berging Spots boven lavabo
bSwitchLight_W3 := bVLight_W3 OR bDK01x1 OR bDK03x1;		//Licht Berging Centraal
bSwitchLight_W4 := bVLight_W4 OR bDK03x4;					//Licht Koele berging
bAllOffBeneden 	:= bDK07x5 OR bDK01x5;

//Melding WC
bMeldingDK02x1 := fbOnOffLight_W1.bLightNormalRelais;

//Licht WC
fbOnOffLight_W1(
	bSwitch:= bSwitchLight_W1,
	bOn:= ,
	bOff:= bAllOff,
	bAutoOff:= TRUE,
	tAutoOffTime:= t#30m,
	bLightNovRam:= bNovRamLight_W1,
	bLightImpulsRelais=> bRelaisLight_W1,
	bLightNormalRelais=> );

//Licht Berging Spots boven lavabo
fbOnOffLight_W2(
	bSwitch:= bSwitchLight_W2,
	bOn:= ,
	bOff:= bAllOffBeneden OR bAllOff,
	bAutoOff:= TRUE,
	tAutoOffTime:= t#15m,
	bLightNovRam:= bNovRamLight_W2,
	bLightImpulsRelais=> bRelaisLight_W2,
	bLightNormalRelais=> );

//Licht Berging Centraal
fbOnOffLight_W3(
	bSwitch:= bSwitchLight_W3,
	bOn:= (P_Doors.ftContactZijdeur.Q AND bAdsSunIsDown),
	bOff:= bAllOffBeneden OR bAllOff,
	bAutoOff:= TRUE,
	tAutoOffTime:= t#15m,
	bLightNovRam:= bNovRamLight_W3,
	bLightImpulsRelais=> bRelaisLight_W3,
	bLightNormalRelais=> );

//Licht Koele berging
fbOnOffLight_W4(
	bSwitch:= bSwitchLight_W4,
	bOn:= ,
	bOff:= bAllOffBeneden OR bAllOff,
	bAutoOff:= TRUE,
	tAutoOffTime:= t#1h,
	bLightNovRam:= bNovRamLight_W4,
	bLightImpulsRelais=> bRelaisLight_W4,
	bLightNormalRelais=> );

END_PROGRAM

// ---- POUs/03-Verlichting/P_LightsBoven.TcPOU
PROGRAM P_LightsBoven
VAR
	(*bSwitchLight_J1: BOOL;*)
	(*bSwitchLight_J2: BOOL;*)
	bSwitchLight_J3		: BOOL;
	bSwitchLight_J4		: BOOL;
	bSwitchLight_W5		: BOOL;
	bSwitchLight_W6		: BOOL;
	bSwitchLight_W7		: BOOL;
	bSwitchLight_W8		: BOOL;
	bSwitchLight_BD2	: BOOL;
	bSwitchLight_BD3	: BOOL;
	bSwitchLight_BD4	: BOOL;
	bSwitchLight_BD5	: BOOL;
	bSwitchLight_BD6	: BOOL;

	bDimLightUp_J3		: BOOL;
	bDimLightDn_J3		: BOOL;
	bSetDimValue_J3		: BOOL;
	uiDimValue_J3		: UINT := 32767;
	tpDoubleTap_J3		: TP;
	iDoubleTap_J3		: INT := 0;

	uiDimValue_BD1		: UINT := 7000;
	uiDimValue_J1		: UINT := 7000;
	uiDimValue_J2		: UINT := 7000;

	//fbOnOffLight_J1		: FB_OnOffLight;
	(*fbOnOffLight_J2	: FB_OnOffLight;*)
	fbOnOffLight_J3		: FB_OnOffLight;
	fbOnOffLight_J4		: FB_OnOffLight;
	fbOnOffLight_W5		: FB_OnOffLight;
	fbOnOffLight_W6		: FB_OnOffLight;
	fbOnOffLight_W7		: FB_OnOffLight;
	fbOnOffLight_W8		: FB_OnOffLight;
	fbOnOffLight_BD2	: FB_OnOffLight;
	fbOnOffLight_BD3	: FB_OnOffLight;
	fbOnOffLight_BD4	: FB_OnOffLight;
	fbOnOffLight_BD5	: FB_OnOffLight;
	fbOnOffLight_BD6	: FB_OnOffLight;
END_VAR


(* Verdiep *)
//bSwitchLight_J1 := bVLight_J1 OR bDK16x1;									//Licht Slaapkamer 3
//bSwitchLight_J2 := bVLight_J2 OR bDK15x1;									//Licht Slaapkamer 2
bSwitchLight_J3 := bVLight_J3 OR bDK14x1 OR bDK13x1;						//Licht Doorgang naar slaapkamer 1 Centraal
bSwitchLight_J4 := bVLight_J4 OR bDK13x2;									//Licht Spots doorgang aan kleerkast
bSwitchLight_W5 := bVLight_W5 OR bDK12x2;									//Licht Douche
(*bSwitchLight_W6 := bSwitchLight_W7;	*)									//Niet in gebruik
bSwitchLight_W7 := bVLight_W7 OR bDK11x3 OR bDK12x1;						//Licht Centraal Badkamer + WC
bSwitchLight_W8 := bVLight_W8 OR bDK11x4;									//Licht Technische Ruimte

bSwitchLight_BD2 := bDK17x3 OR bDK19x1 OR bDK20x1;							//Licht kleerkast Slaapkamer 1
bSwitchLight_BD3 := bDK17x4 OR bDK19x2 OR bDK20x2;							//Licht dressoir Slaapkamer 1
bSwitchLight_BD4 := bDK21x2;												//Licht bad
bSwitchLight_BD5 := bDK21x1 OR bDK22x1;										//Licht badkamer 2

//Melding
bMeldingDK11x3 := bNovRamLight_W5 OR bNovRamLight_W7;
bMeldingDK11x4 := bNovRamLight_W8;

//Dimmer Slaapkamer 3
fbDimmer_J1(
	bSwitchDimmUp:= bDK16x1,
	bSwitchDimmDown:= bDK16x2,
	bOn:=  ,
	bOff:= bAllOff,
	bSwitchSetpUp := ,
	bSwitchSetpDown := ,
	bSetDimmValue:=  ,
	nDimmValue:= uiDimValue_J1,
	tSwitchOverTime:= t#400ms,
	tDimmTime:= tDimmerTijd,
	bMemoryModeOn:= TRUE,
	nOnValueWithoutMemoryMode:= ,
	bDimmOnMode:= ,
	tDimmOnTime:= ,
	bDimmOffMode:= ,
	tDimmOffTime:= ,
	nOutMin:= 3500,
	nOutMax:= 32767,
	nSavedOut := nDimmValue_J1,
	nOut=> DimLight_J1,
	bLight=> );

//Dimmer Slaapkamer 2
fbDimmer_J2(
	bSwitchDimmUp:= bDK15x1,
	bSwitchDimmDown:= bDK15x2,
	bOn:=  ,
	bOff:= bAllOff,
	bSwitchSetpUp := ,
	bSwitchSetpDown := ,
	bSetDimmValue:=  ,
	nDimmValue:= uiDimValue_J2,
	tSwitchOverTime:= t#400ms,
	tDimmTime:= tDimmerTijd,
	bMemoryModeOn:= TRUE,
	nOnValueWithoutMemoryMode:= ,
	bDimmOnMode:= ,
	tDimmOnTime:= ,
	bDimmOffMode:= ,
	tDimmOffTime:= ,
	nOutMin:= 3500,
	nOutMax:= 32767,
	nSavedOut := nDimmValue_J2,
	nOut=> DimLight_J2,
	bLight=> );

//Licht Doorgang naar slaapkamer 1 Centraal
fbOnOffLight_J3(
	bSwitch:= bSwitchLight_J3,
	bOn:= ,
	bOff:= bAllOff,
	bAutoOff:= ,
	tAutoOffTime:= ,
	bLightNovRam:= bNovRamLight_J3,
	bLightImpulsRelais=> bRelaisLight_J3,
	bLightNormalRelais=> );

//Licht Spots doorgang aan kleerkast
fbOnOffLight_J4(
	bSwitch:= bSwitchLight_J4,
	bOn:= ,
	bOff:= bAllOff,
	bAutoOff:= ,
	tAutoOffTime:= ,
	bLightNovRam:= bNovRamLight_J4,
	bLightImpulsRelais=> bRelaisLight_J4,
	bLightNormalRelais=> );

//Licht Douche
fbOnOffLight_W5(
	bSwitch:= bSwitchLight_W5,
	bOn:= ,
	bOff:= bAllOff,
	bAutoOff:= ,
	tAutoOffTime:= ,
	bLightNovRam:= bNovRamLight_W5,
	bLightImpulsRelais=> bRelaisLight_W5,
	bLightNormalRelais=> );

fbOnOffLight_W6(
	bSwitch:= ,
	bOn:= ,
	bOff:= ,
	bAutoOff:= ,
	tAutoOffTime:= ,
	bLightNovRam:= bNovRamLight_W6,
	bLightImpulsRelais=> bRelaisLight_W6,
	bLightNormalRelais=> );

//Licht Centraal Badkamer + WC
fbOnOffLight_W7(
	bSwitch:= bSwitchLight_W7,
	bOn:= ,
	bOff:= bAllOff,
	bAutoOff:= ,
	tAutoOffTime:= ,
	bLightNovRam:= bNovRamLight_W7,
	bLightImpulsRelais=> bRelaisLight_W7,
	bLightNormalRelais=> );
bRelaisLight_W6 := bRelaisLight_W7;

//Licht Technische Ruimte
fbOnOffLight_W8(
	bSwitch:= bSwitchLight_W8,
	bOn:= ,
	bOff:= bAllOff,
	bAutoOff:= ,
	tAutoOffTime:= ,
	bLightNovRam:= bNovRamLight_W8,
	bLightImpulsRelais=> bRelaisLight_W8,
	bLightNormalRelais=> );

//Licht kleerkast Slaapkamer 1
fbOnOffLight_BD2(
	bSwitch:= bSwitchLight_BD2,
	bOn:= ,
	bOff:= bAllOff,
	bAutoOff:= ,
	tAutoOffTime:= ,
	bLightNovRam:= bNovRamLight_BD2,
	bLightImpulsRelais=> bRelaisLight_BD2,
	bLightNormalRelais=> );

//Licht dressoir Slaapkamer 1
fbOnOffLight_BD3(
	bSwitch:= bSwitchLight_BD3,
	bOn:= ,
	bOff:= bAllOff,
	bAutoOff:= ,
	tAutoOffTime:= ,
	bLightNovRam:= bNovRamLight_BD3,
	bLightImpulsRelais=> bRelaisLight_BD3,
	bLightNormalRelais=> );

//Licht bad
fbOnOffLight_BD4(
	bSwitch:= bSwitchLight_BD4,
	bOn:= ,
	bOff:= bAllOff,
	bAutoOff:= ,
	tAutoOffTime:= ,
	bLightNovRam:= bNovRamLight_BD4,
	bLightImpulsRelais=> bRelaisLight_BD4,
	bLightNormalRelais=> );

//Licht badkamer 2
fbOnOffLight_BD5(
	bSwitch:= bSwitchLight_BD5,
	bOn:= ,
	bOff:= bAllOff,
	bAutoOff:= ,
	tAutoOffTime:= ,
	bLightNovRam:= bNovRamLight_BD5,
	bLightImpulsRelais=> bRelaisLight_BD5,
	bLightNormalRelais=> );


//Dimmer Slaapkamer 1 Centraal
fbDimmer_BD1(
	bSwitchDimmUp:= bDK17x1 OR bDK18x1 OR bDK13x4,
	bSwitchDimmDown:= bDK17x2 OR bDK18x2,
	bOn:= ,
	bOff:= bAllOff,
	bSwitchSetpUp := ,
	bSwitchSetpDown := ,
	bSetDimmValue:=  ,
	nDimmValue:= uiDimValue_BD1,
	tSwitchOverTime:= t#400ms,
	tDimmTime:= tDimmerTijd,
	bMemoryModeOn:= TRUE,
	nOnValueWithoutMemoryMode:= ,
	bDimmOnMode:= ,
	tDimmOnTime:= ,
	bDimmOffMode:= ,
	tDimmOffTime:= ,
	nOutMin:= 3500,
	nOutMax:= 32767,
	nSavedOut := nDimmValue_BD1,
	nOut=> DimLight_BD1,
	bLight=> );

END_PROGRAM

// ---- POUs/03-Verlichting/P_LightsBuiten.TcPOU
PROGRAM P_LightsBuiten
VAR
	bSwitchLight_Y4		: BOOL;
	bSwitchLight_Y6		: BOOL;
	bSwitchLight_Y7		: BOOL;
	bSwitchLight_Z1		: BOOL;
	bSwitchLight_Z2		: BOOL;
	bSwitchLight_Z3		: BOOL;
	bSwitchLight_Z4		: BOOL;
	bSwitchLight_BD8	: BOOL;

	fbOnOffLight_Y4		: FB_OnOffLight;
	fbOnOffLight_Y6		: FB_OnOffLight;
	fbOnOffLight_Y7		: FB_OnOffLight;

	fbOnOffLight_Z1		: FB_OnOffLight;
	fbOnOffLight_Z2		: FB_OnOffLight;
	fbOnOffLight_Z3		: FB_OnOffLight;
	fbOnOffLight_Z4		: FB_OnOffLight;
	fbOnOffLight_BD8	: FB_OnOffLight;

	bAutoOffBD8			: BOOL := TRUE;

	(* Tuinhuis achteraan *)
	bSwitchLight_ZZ1	: BOOL;
	bSwitchLight_ZZ2	: BOOL;
	fbOnOffLight_ZZ1	: FB_OnOffLight;
	fbOnOffLight_ZZ2	: FB_OnOffLight;
END_VAR


bSwitchLight_Z1 := bVLight_Z1 OR bDK30x1;					//Licht TL Tuinhuis
bSwitchLight_Z2 := bVLight_Z2;								//Licht Led spots frame Tuinhuis
bSwitchLight_Z3 := bVLight_Z3 OR bDK01x2 OR bDK10x3;		//Licht Vuilbakken
bSwitchLight_Z4 := bVLight_Z4;								//Geschakeld stopcontact tuinhuis. Controleren of nog in gebruik
bSwitchLight_BD8 := bDK10x4 OR bDK19x4;						//2 Spots buitengevel leefruimte voor terras
bSwitchLight_ZZ1 := bDK40x2;								//2 spots aan wand tuinhuis achteraan
bSwitchLight_ZZ2 := bDK40x1 OR bDK10x2; 					//Centrale spots tuinhuis achteraan

//Spots carport
fbOnOffLight_Y4(
	bSwitch:= bSwitchLight_Y4,
	bOn:= (P_Doors.ftContactZijdeur.Q AND bAdsSunIsDown),
	bOff:= ,
	bAutoOff:= TRUE,
	tAutoOffTime:= T#2M,
	bLightNovRam:= bNovRamLight_Y4,
	bLightImpulsRelais=> bRelaisLight_Y4);

//Up/Down spots voorgevel huis
fbOnOffLight_Y7(
	bSwitch:= bSwitchLight_Y7,
	bOn:= P_SunriseSunset.bSunsetPulse,
	bOff:= P_SunriseSunset.bSunrisePulse,
	bAutoOff:= ,
	tAutoOffTime:= ,
	bLightNovRam:= bNovRamLight_Y7,
	bLightImpulsRelais=> bRelaisLight_Y7);

//TL Tuinhuis
fbOnOffLight_Z1(
	bSwitch:= bSwitchLight_Z1,
	bOn:= ,
	bOff:= bAllOff,
	bAutoOff:= ,
	tAutoOffTime:= ,
	bLightNovRam:= bNovRamLight_Z1,
	bLightImpulsRelais=> bRelaisLight_Z1);

//Licht Led spots frame Tuinhuis
fbOnOffLight_Z2(
	bSwitch:= bSwitchLight_Z2,
	bOn:= P_SunriseSunset.bSunsetPulse,
	bOff:= P_SunriseSunset.bSunrisePulse,
	bAutoOff:= ,
	tAutoOffTime:= ,
	bLightNovRam:= bNovRamLight_Z2,
	bLightImpulsRelais=> bRelaisLight_Z2);

//Licht Vuilbakken
fbOnOffLight_Z3(
	bSwitch:= bSwitchLight_Z3,
	bOn:= ,
	bOff:= bAllOff,
	bAutoOff:= TRUE,
	tAutoOffTime:= t#10m,
	bLightNovRam:= bNovRamLight_Z3,
	bLightImpulsRelais=> bRelaisLight_Z3 );

//Geschakeld stopcontact
fbOnOffLight_Z4(
	bSwitch:= bSwitchLight_Z4,
	bOn:= ,
	bOff:= bAllOff,
	bAutoOff:= ,
	tAutoOffTime:= ,
	bLightNovRam:= bNovRamLight_Z4,
	bLightImpulsRelais=> bRelaisLight_Z4 );

//2 Spots buitengevel leefruimte voor terras
fbOnOffLight_BD8(
	bSwitch:= bSwitchLight_BD8,
	bOn:= ,
	bOff:= bAllOff,
	bAutoOff:= bAutoOffBD8,
	tAutoOffTime:= t#1m,
	bSensorActivation := (*bSensTuinhuisBuiten AND bAutoOffBD8 AND (todWinTime > (todZonOnder - T#30m)) AND (todWinTime < TOD#23:00:00)(* OR todWinTime < (todZonOp + T#25m))*)  *),
	bLightNovRam:= bNovRamLight_BD8,
	bLightNormalRelais=> bRelaisLight_BD8 );

//Stopcontact robotmaaier
fbOnOffLight_Y6(
	bSwitch:= bSwitchLight_Y6,
	bOn:= (*bSunsetOn*),
	bOff:= (*bAllOff OR bAllOffBeneden OR bSunriseOff*),
	bAutoOff:= ,
	tAutoOffTime:= ,
	bSensorActivation := ,
	bLightNovRam:= bNovRamLight_Y6,
	bLightImpulsRelais=> bRelaisLight_Y6 );

//2 spots aan wand tuinhuis achteraan
fbOnOffLight_ZZ1(
	bSwitch:= bSwitchLight_ZZ1,
	bOn:= ,
	bOff:= bAllOff OR bAllOffBeneden,
	bAutoOff:= ,
	tAutoOffTime:= ,
	bLightNovRam:= bNovRamLight_ZZ1,
	bLightImpulsRelais=> bRelaisLight_ZZ1);

//Centrale spots tuinhuis achteraan
fbOnOffLight_ZZ2(
	bSwitch:= bSwitchLight_ZZ2,
	bOn:= ,
	bOff:=  bAllOff OR bAllOffBeneden,
	bAutoOff:= ,
	tAutoOffTime:= ,
	bLightNovRam:= bNovRamLight_ZZ2,
	bLightImpulsRelais=> bRelaisLight_ZZ2);

END_PROGRAM

// ---- POUs/03-Verlichting/P_LightsHal.TcPOU
PROGRAM P_LightsHal
VAR
	bSwitchLight_I1	: BOOL;
	bSwitchLight_J5	: BOOL;
	bSwitchLight_J6	: BOOL;

	fbOnOffLight_I1	: FB_OnOffLight;
	fbOnOffLight_J5	: FB_OnOffLight;
	fbOnOffLight_J6	: FB_OnOffLight;
END_VAR


//Hal en Traphal
bSwitchLight_I1 := bVLight_I1 OR bDK08x1;								//Licht Hal
bSwitchLight_J5 := bVLight_J5 OR bDK08x3 OR bDK11x1 OR bDK14x3;			//Licht Spots Traphal plafond
bSwitchLight_J6 := bVLight_J6 OR bDK08x2;								//Licht Spots Traphal wand

//Licht Hal
fbOnOffLight_I1(
	bSwitch:= bSwitchLight_I1,
	(*bOn:=  (P_Doors.ftContactVoordeur.Q AND bZonOnder),*)
	bOff:= bAllOffBeneden OR bAllOff,
	bAutoOff:= ,
	tAutoOffTime:= ,
	bLightNovRam:= bNovRamLight_I1,
	bLightImpulsRelais=> bRelaisLight_I1);

//Licht Spots Traphal plafond
fbOnOffLight_J5(
	bSwitch:= bSwitchLight_J5,
	bOn:= ,
	bOff:= bAllOffBeneden OR bAllOff,
	bAutoOff:= ,
	tAutoOffTime:= ,
	bLightNovRam:= bNovRamLight_J5,
	bLightImpulsRelais=> bRelaisLight_J5);

//Licht Spots Traphal wand
fbOnOffLight_J6(
	bSwitch:= bSwitchLight_J6,
	bOn:= P_SunriseSunset.bSunsetPulse,
	bOff:= P_SunriseSunset.bSunrisePulse,
	bAutoOff:= ,
	tAutoOffTime:= ,
	bLightNovRam:= bNovRamLight_J6,
	bLightImpulsRelais=> bRelaisLight_J6);

END_PROGRAM

// ---- POUs/03-Verlichting/P_LightsKeukenLiving.TcPOU
PROGRAM P_LightsKeukenLiving
VAR
	rtAdsLichtKeukenCentraal		: R_TRIG;
	rtAdsLichtKeukenSpotsDampkap	: R_TRIG;
	rtAdsLichtLivingStepUp			: R_TRIG;
	rtAdsLichtLivingStepDown		: R_TRIG;

	bSwitchLight_I2					: BOOL;
	bSwitchLight_I3					: BOOL;
	bSwitchLight_I4					: BOOL;
	bSwitchLight_I5					: BOOL;
	bSwitchLight_I7					: BOOL;

	bAanwezigKeukenLiving			: BOOL;

	fbOnOffLight_I3					: FB_OnOffLight;
	fbOnOffLight_I5					: FB_OnOffLight;
	fbOnOffLight_I7					: FB_OnOffLight;
	fbOnOffLight_I8					: FB_OnOffLight;

	(* Centrale verlichting Living *)
	bDimLightUp_I2					: BOOL;
	bDimLightDn_I2					: BOOL;
	bSetDimValue_I2					: BOOL;
	uiDimValue_I2					: UINT := 7000;
END_VAR

rtAdsLichtKeukenCentraal(CLK:=bAdsLichtKeukenCentraal);
rtAdsLichtKeukenSpotsDampkap(CLK:=bAdsLichtKeukenSpotsDampkap);
rtAdsLichtLivingStepUp(CLK:=bAdsLichtLivingStepUp);
rtAdsLichtLivingStepDown(CLK:=bAdsLichtLivingStepDown);

bSwitchLight_I3 := bVLight_I3 OR bDK07x3;																	//Geschakeld Stopcontact hoek Living (K3)
bSwitchLight_I4 := bVLight_I4;																				//Button+ Altijd aan
bSwitchLight_I5 := bVLight_I5 OR bDK04x1 OR bDK05x1 OR bDK07x4 OR bDK03x2 OR rtAdsLichtKeukenCentraal.Q;	//Licht Kookeiland Centraal
bSwitchLight_I7 := bVLight_I7 OR bDK05x2 OR rtAdsLichtKeukenSpotsDampkap.Q;									//Licht Spots Dampkap

//Aanwezigheid
bAanwezigKeukenLiving := bNovRamLight_I3 OR bNovRamLight_I4 OR bNovRamLight_I5 OR bNovRamLight_I7 OR fbDimmer_I2.bLight;

//Geschakeld Stopcontact hoek Living (K3)
fbOnOffLight_I3(
	bSwitch:= bSwitchLight_I3,
	bOn:= ,
	bOff:= bAllOff OR bAllOffBeneden,
	bAutoOff:= ,
	tAutoOffTime:= ,
	bLightNovRam:= bNovRamLight_I3,
	bLightImpulsRelais=> bRelaisLight_I3);

//Licht Kookeiland Centraal
fbOnOffLight_I5(
	bSwitch:= bSwitchLight_I5 ,
	bOn:= (* OR (P_Doors.ftContactSchuifdeurLeefruimte.Q AND bZonOnder AND NOT bAanwezigKeukenLiving)*),
	bOff:= bAllOff OR bAllOffBeneden,
	bAutoOff:= ,
	tAutoOffTime:= ,
	bLightNovRam:= bNovRamLight_I5,
	bLightImpulsRelais=> bRelaisLight_I5);

//Licht Spots Dampkap
fbOnOffLight_I7(
	bSwitch:= bSwitchLight_I7,
	bOn:= ,
	bOff:= bAllOff OR bAllOffBeneden,
	bAutoOff:= ,
	tAutoOffTime:= ,
	bLightNovRam:= bNovRamLight_I7,
	bLightImpulsRelais=> bRelaisLight_I7);


//Dimmer Living centraal
bDimLightUp_I2 := bVLight_I2 OR bDK07x1;
bDimLightDn_I2 := bDK07x2;

fbDimmer_I2(
	bSwitchDimmUp:= bDimLightUp_I2,
	bSwitchDimmDown:= bDimLightDn_I2,
	bOn:=  ,
	bOff:= bAllOff OR bAllOffBeneden,
	bSwitchSetpUp := rtAdsLichtLivingStepUp.Q,
	bSwitchSetpDown := rtAdsLichtLivingStepDown.Q,
	bSetDimmValue:= bSetDimValue_I2 ,
	nDimmValue:= uiDimValue_I2,
	tSwitchOverTime:= t#400ms,
	tDimmTime:= tDimmerTijd,
	bMemoryModeOn:= TRUE,
	nOnValueWithoutMemoryMode:= ,
	bDimmOnMode:= ,
	tDimmOnTime:= ,
	bDimmOffMode:= ,
	tDimmOffTime:= ,
	nOutMin:= 3500,
	nOutMax:= 27000,
	nSavedOut := nDimmValue_I2,
	nOut=> DimLight_I2,
	bLight=> );

END_PROGRAM

// ---- POUs/03-Verlichting/P_LightsLeefruimte.TcPOU
PROGRAM P_LightsLeefruimte
VAR
	bSwitchLight_Y1	: BOOL;
	bSwitchLight_Y2	: BOOL;
	bSwitchLight_Y3	: BOOL;
(*	bSwitchLight_Y4	: BOOL;
	bSwitchLight_Y5	: BOOL;
	bSwitchLight_Y6	: BOOL;
	bSwitchLight_Y7	: BOOL; *)


	fbOnOffLight_Y1	: FB_OnOffLight;
	fbOnOffLight_Y2	: FB_OnOffLight;
	fbOnOffLight_Y3	: FB_OnOffLight;
	fbOnOffLight_Y5	: FB_OnOffLight;

END_VAR


bSwitchLight_Y1 := bVLight_Y1 OR bDK09x3;						//Leefruimte Spots Barkast
bSwitchLight_Y2 := bVLight_Y2 OR bDK09x1 OR bDK10x1 OR bDK04x2;	//Leefruimte Centraal eettafel
bSwitchLight_Y3 := bVLight_Y3 OR bDK09x2;						//Leefruimte Spots zithoek

//Leefruimte Spots Barkast
fbOnOffLight_Y1(
	bSwitch:= bSwitchLight_Y1,
	bOn:= ,
	bOff:= bAllOffBeneden OR bAllOff,
	bAutoOff:= ,
	tAutoOffTime:= ,
	bLightNovRam:= bNovRamLight_Y1,
	bLightImpulsRelais=> bRelaisLight_Y1);

//Leefruimte Centraal eettafel
fbOnOffLight_Y2(
	bSwitch:= bSwitchLight_Y2,
	bOn:= ,
	bOff:= bAllOffBeneden OR bAllOff,
	bAutoOff:= ,
	tAutoOffTime:= ,
	bLightNovRam:= bNovRamLight_Y2,
	bLightImpulsRelais=> bRelaisLight_Y2);

//Leefruimte Spots zithoek
fbOnOffLight_Y3(
	bSwitch:= bSwitchLight_Y3,
	bOn:= ,
	bOff:= bAllOffBeneden OR bAllOff,
	bAutoOff:= ,
	tAutoOffTime:= ,
	bLightNovRam:= bNovRamLight_Y3,
	bLightImpulsRelais=> bRelaisLight_Y3);

//Up/Down spots muur leefruimte
fbOnOffLight_Y5(
	bSwitch:= ,
	bOn:= P_SunriseSunset.bSunsetPulse,
	bOff:= P_SunriseSunset.bSunrisePulse OR bAllOffBeneden,
	bAutoOff:= ,
	tAutoOffTime:= ,
	bLightNovRam:= bNovRamLight_Y5,
	bLightImpulsRelais=> bRelaisLight_Y5);

END_PROGRAM

// ---- POUs/04-Boiler/P_Boiler.TcPOU
PROGRAM P_Boiler
VAR
	bBoilerOn		: BOOL;
	bBoilerOff		: BOOL;
	bVBoilerSwitch	: BOOL;
	fbOnOffBoiler	: FB_OnOffLight;
END_VAR

fbOnOffBoiler(
	bSwitch:= bVBoilerSwitch OR bAdsBoilerOnOff,
	bOn:= bBoilerOn OR (todWinTime = tod#13:00 AND P_Temperatures.rTempBoiler < 55),
	bOff:= bBoilerOff,
	bAutoOff:= TRUE,
	tAutoOffTime:= t#4h,
	bLightNovRam:= bNovRamBoiler,
	bLightImpulsRelais=> bRelaisBoiler);

bAdsBoilerState := bNovRamBoiler;

END_PROGRAM

// ---- POUs/05-Temperaturen/P_Temperatures.TcPOU
PROGRAM P_Temperatures
VAR
	rTempKeuken: REAL;
	rTempLiving: REAL;
	rTempBoiler: REAL;
END_VAR

rTempBoiler := INT_TO_REAL(iTemp6) / 100;
rTempLiving := INT_TO_REAL(iTemp7) / 100;
rTempKeuken := INT_TO_REAL(iTemp8) / 100;

END_PROGRAM

// ---- POUs/06-Screens/P_Screens.TcPOU
PROGRAM P_Screens
VAR
	bScreen1Omhoog				: BOOL;
	bScreen1Omlaag				: BOOL;
	bScreen2Omhoog				: BOOL;
	bScreen2Omlaag				: BOOL;
	bScreen3Omhoog				: BOOL;
	bScreen3Omlaag				: BOOL;
	bScreen4Omhoog				: BOOL;
	bScreen4Omlaag				: BOOL;
	bRolluik1Omhoog				: BOOL;
	bRolluik1Omlaag				: BOOL;
	bRolluik2Omhoog				: BOOL;
	bRolluik2Omlaag				: BOOL;
	bRolluik3Omhoog				: BOOL;
	bRolluik3Omlaag				: BOOL;

	fbScreen1					: FB_Screens;
	fbScreen2					: FB_Screens;
	fbScreen3					: FB_Screens;
	fbScreen4					: FB_Screens;
	fbRolluik1					: FB_Screens;
	fbRolluik2					: FB_Screens;
	fbRolluik3					: FB_Screens;

	bAutomaticScreens			: BOOL;
	rtAutomaticScreens			: R_TRIG;

	bBeveiligingHogeWindsnelheidActief	: BOOL;

	tpAutomaticScreen123Up		: TP;
	tpAutomaticScreen123Dn		: TP;
	tpAutomaticScreen4Up		: TP;
	tpAutomaticScreen4Dn		: TP;
	tpAutomaticRolluik1Dn		: TP;
	tpAutomaticRolluik2Dn		: TP;
	tpAutomaticRolluik3Dn		: TP;
END_VAR

bScreen1Omhoog := bDK04x3 (*OR tpAutomaticScreen123Up.Q*);
bScreen1Omlaag := bDK04x4 (*OR (tpAutomaticScreen123Dn.Q AND bAutomaticScreens)*);
bScreen2Omhoog := bDK10x5 (*OR tpAutomaticScreen123Up.Q*);
bScreen2Omlaag := bDK10x6 (*OR tpAutomaticScreen123Dn.Q*);
bScreen3Omhoog := bDK04x3 (*OR tpAutomaticScreen123Up.Q*);
bScreen3Omlaag := bDK04x4 (*OR (tpAutomaticScreen123Dn.Q AND bAutomaticScreens)*);
bScreen4Omhoog := bDK04x5 (*OR tpAutomaticScreen4Up.Q*);
bScreen4Omlaag := bDK04x6 (*OR (tpAutomaticScreen4Dn.Q AND bAutomaticScreens)*);


bRolluik1Omhoog := bDK17x5 OR bDK18x3 OR bDK19x5;
bRolluik1Omlaag := bDK17x6 OR bDK18x4 OR bDK19x6 OR (tpAutomaticRolluik1Dn.Q AND bAutomaticScreens);
bRolluik2Omhoog := bDK16x3 ;
bRolluik2Omlaag := bDK16x4 OR (tpAutomaticRolluik2Dn.Q AND bAutomaticScreens);
bRolluik3Omhoog := bDK15x3 ;
bRolluik3Omlaag := bDK15x4 OR (tpAutomaticRolluik3Dn.Q AND bAutomaticScreens);

(* Screen Links van Schuifraam *)
fbScreen1(
	bUp:=  bAdsScreen13Up OR bAdsAllScreensUp,
	bDown:= bAdsScreen13Dn OR bAdsAllScreensDn,
	bStop:=  ,
	bSwitchOverUp:= bScreen1Omhoog ,
	bSwitchOverDown:= bScreen1Omlaag ,
	tSwitchOverTime:= t#500ms,
	bStepUp:= ,
	bStepDown:= ,
	tStepTime:= ,
	bShadowPosition:= ,
	tShadowTurnAroundTime:= ,
	tShadowTurnOffTime:= ,
	bSafetyPosition:= (*P_Windmeter.bHogeWindsnelheid AND *) bBeveiligingHogeWindsnelheidActief,
	tTurnOffTime:= t#22s,
	tSwitchOverDeadTime:= t#1s,
	bBlindUp=> bMotorScreen1Omhoog,
	bBlindDown=> bMotorScreen1Omlaag );

(* Screen Schuifraam *)
fbScreen2(
	bUp:= (*fbShortLongClick30x1.bLongPress1 OR*) bAdsScreen2Up OR bAdsAllScreensUp,
	bDown:= bAdsScreen2Dn OR bAdsAllScreensDn,
	bStop:=  ,
	bSwitchOverUp:= bScreen2Omhoog ,
	bSwitchOverDown:= bScreen2Omlaag ,
	tSwitchOverTime:= t#500ms,
	bStepUp:= ,
	bStepDown:= ,
	tStepTime:= ,
	bShadowPosition:= ,
	tShadowTurnAroundTime:= ,
	tShadowTurnOffTime:= ,
	bSafetyPosition:= (*P_Windmeter.bHogeWindsnelheid AND *) bBeveiligingHogeWindsnelheidActief,
	tTurnOffTime:= t#22s,
	tSwitchOverDeadTime:= t#1s,
	bBlindUp=> bMotorScreen2Omhoog,
	bBlindDown=> bMotorScreen2Omlaag );

(* Screen Rechts van Schuifraam *)
fbScreen3(
	bUp:= bAdsScreen13Up OR bAdsAllScreensUp,
	bDown:= bAdsScreen13Dn OR bAdsAllScreensDn,
	bStop:=  ,
	bSwitchOverUp:= bScreen3Omhoog ,
	bSwitchOverDown:= bScreen3Omlaag ,
	tSwitchOverTime:= t#500ms,
	bStepUp:= ,
	bStepDown:= ,
	tStepTime:= ,
	bShadowPosition:= ,
	tShadowTurnAroundTime:= ,
	tShadowTurnOffTime:= ,
	bSafetyPosition:= (*P_Windmeter.bHogeWindsnelheid AND *) bBeveiligingHogeWindsnelheidActief,
	tTurnOffTime:= t#22s,
	tSwitchOverDeadTime:= t#1s,
	bBlindUp=> bMotorScreen3Omhoog,
	bBlindDown=> bMotorScreen3Omlaag );

(* Screen lange venster *)
fbScreen4(
	bUp:= bAdsScreen4Up OR bAdsAllScreensUp,
	bDown:= bAdsScreen4Dn OR bAdsAllScreensDn,
	bStop:=  ,
	bSwitchOverUp:= bScreen4Omhoog ,
	bSwitchOverDown:= bScreen4Omlaag ,
	tSwitchOverTime:= t#500ms,
	bStepUp:= ,
	bStepDown:= ,
	tStepTime:= ,
	bShadowPosition:= ,
	tShadowTurnAroundTime:= ,
	tShadowTurnOffTime:= ,
	bSafetyPosition:= (*P_Windmeter.bHogeWindsnelheid AND *) bBeveiligingHogeWindsnelheidActief,
	tTurnOffTime:= t#8s,
	tSwitchOverDeadTime:= t#1s,
	bBlindUp=> bMotorScreen4Omhoog,
	bBlindDown=> bMotorScreen4Omlaag );

(* Rolluik Slaapkamer mama papa *)
fbRolluik1(
	bUp:= ,
	bDown:= ,
	bStop:=  ,
	bSwitchOverUp:= bRolluik1Omhoog ,
	bSwitchOverDown:= bRolluik1Omlaag ,
	tSwitchOverTime:= t#500ms,
	bStepUp:= ,
	bStepDown:= ,
	tStepTime:= ,
	bShadowPosition:= ,
	tShadowTurnAroundTime:= ,
	tShadowTurnOffTime:= ,
	bSafetyPosition:= ,
	tTurnOffTime:= t#27s,
	tSwitchOverDeadTime:= t#1s,
	bBlindUp=> bMotorRolluik1Omhoog,
	bBlindDown=> bMotorRolluik1Omlaag );


(* Rolluik Slaapkamer Lukas *)
fbRolluik2(
	bUp:= ,
	bDown:= ,
	bStop:=  ,
	bSwitchOverUp:= bRolluik2Omhoog ,
	bSwitchOverDown:= bRolluik2Omlaag ,
	tSwitchOverTime:= t#500ms,
	bStepUp:= ,
	bStepDown:= ,
	tStepTime:= ,
	bShadowPosition:= ,
	tShadowTurnAroundTime:= ,
	tShadowTurnOffTime:= ,
	bSafetyPosition:= ,
	tTurnOffTime:= t#27s,
	tSwitchOverDeadTime:= t#1s,
	bBlindUp=> bMotorRolluik2Omhoog,
	bBlindDown=> bMotorRolluik2Omlaag );


(* Rolluik Slaapkamer Elena *)
fbRolluik3(
	bUp:= ,
	bDown:= ,
	bStop:=  ,
	bSwitchOverUp:= bRolluik3Omhoog ,
	bSwitchOverDown:= bRolluik3Omlaag ,
	tSwitchOverTime:= t#500ms,
	bStepUp:= ,
	bStepDown:= ,
	tStepTime:= ,
	bShadowPosition:= ,
	tShadowTurnAroundTime:= ,
	tShadowTurnOffTime:= ,
	bSafetyPosition:= ,
	tTurnOffTime:= t#27s,
	tSwitchOverDeadTime:= t#1s,
	bBlindUp=> bMotorRolluik3Omhoog,
	bBlindDown=> bMotorRolluik3Omlaag );

END_PROGRAM

// ---- POUs/07-Draaipoort/P_Draaipoort.TcPOU
PROGRAM P_Draaipoort
VAR
	tonDraaipoortVolledig		: TON;
	tpDraaipoortVolledig		: TP;

	tonDraaipoortVoetganger		: TON;
	tpDraaipoortVoetganger		: TP;
END_VAR

tonDraaipoortVolledig(IN:= bDK01x4 OR bAdsPoortOpenDicht, PT:= T#500MS, Q=> , ET=> );
tpDraaipoortVolledig(IN:= tonDraaipoortVolledig.Q, PT:= t#500ms, Q=> bDraaipoortVolledigOpenDicht, ET=> );


tonDraaipoortVoetganger(IN:= bDK01x3 OR bAdsPoortVoetganger, PT:= t#500ms, Q=> , ET=> );
tpDraaipoortVoetganger(IN:= tonDraaipoortVoetganger.Q, PT:= t#500ms, Q=> bDraaipoortVoetgangerOpenDicht, ET=> );

END_PROGRAM

// ---- POUs/08-Energiemetingen/P_Kwartierpiek.TcPOU
PROGRAM P_Kwartierpiek
VAR
	todSystemTime						: TOD;
                            		
	todStartTime						: TOD;
	CurrentActivePower					: REAL;
	iWhMeter							: DINT;
	iStartWhMeter						: DINT;
	tRestTijd							: TIME;
                            			
	rKwartuurVoorspelling1				: REAL;
	rKwartuurVoorspelling2				: REAL;
	rKwartuurVoorspelling3				: REAL;

	tonDelayKwartuur					: TON;
	bMaximaleKwartuurpiekOverschreiding : BOOL;
	rStandaardActiefVermogen			: REAL := 600; (*kW*)
	rMaximaleKwartuurpiek				: REAL := 3500; (*kW*)
	rGewenstActiefVermogen				: REAL;
	tVerstrekenTijd						: TIME;

	sOverKwartierpiek					: STRING;

END_VAR

(* Voorspelling kwartuurpiek*)
todSystemTime := DT_TO_TOD(SYSTEMTIME_TO_DT(strWinTime));

IF (strWinTime.wMinute MOD 15) = 0 AND strWinTime.wSecond = 0 THEN
	todStartTime := todSystemTime;
	iStartWhMeter := iWhMeter;
END_IF

IF (iStartWhMeter <> 0) THEN
	tRestTijd := (todStartTime - todSystemTime) + T#15M;
	IF tRestTijd > t#15M THEN
		tRestTijd := t#15M;
	END_IF
	tVerstrekenTijd := t#15M - tRestTijd;

	rKwartuurVoorspelling1 := (iWhMeter - iStartWhMeter)*4.0;  (* Eerste berekening. Gebruikte kWh * 4 = kwartuurpiek als er vanaf dan 0W actief vermogen zou zijn *)
	rKwartuurVoorspelling2 := rKwartuurVoorspelling1 + (CurrentActivePower*TIME_TO_REAL(tRestTijd)/900000); (* Eerste berekening + Als huidig actief vermogen zou aangehouden worden voor resterende tijd *)

	IF TIME_TO_REAL(tVerstrekenTijd) > 0 THEN
		rKwartuurVoorspelling3 := (iWhMeter - iStartWhMeter) * (60/ (TIME_TO_REAL(tVerstrekenTijd)/60000)); (* Extrapolatie van kWh meterstand gelet op de verstreken tijd. Delen door 60000 voor omzetting naar minuten*)
	END_IF


	tonDelayKwartuur(IN:= rKwartuurVoorspelling2 > rMaximaleKwartuurpiek, PT:=t#1m, Q=> bMaximaleKwartuurpiekOverschreiding);
	IF (rKwartuurVoorspelling2 > rMaximaleKwartuurpiek) AND (TIME_TO_REAL(tRestTijd)/900000 > 0) THEN
		rGewenstActiefVermogen := (rMaximaleKwartuurpiek - rKwartuurVoorspelling1) / (TIME_TO_REAL(tRestTijd)/900000);
		IF rGewenstActiefVermogen < 0 THEN
			rGewenstActiefVermogen := 0;
		ELSIF rGewenstActiefVermogen > 3000 THEN
			rGewenstActiefVermogen := 3000;
		END_IF
	ELSE
		rGewenstActiefVermogen := rMaximaleKwartuurpiek;
	END_IF
END_IF

IF bMaximaleKwartuurpiekOverschreiding THEN
	sOverKwartierpiek := CONCAT('Verlaag vermogen naar ', UDINT_TO_STRING(REAL_TO_UDINT(rGewenstActiefVermogen)));
	sOverKwartierpiek := CONCAT(sOverKwartierpiek, 'W, voorspelde piek ');
	sOverKwartierpiek := CONCAT(sOverKwartierpiek, UDINT_TO_STRING(REAL_TO_UDINT(rKwartuurVoorspelling2)));
	sOverKwartierpiek := CONCAT(sOverKwartierpiek, 'W, resterende tijd ');
	sOverKwartierpiek := CONCAT(sOverKwartierpiek, UDINT_TO_STRING(TIME_TO_UDINT(tRestTijd)/1000));
	sOverKwartierpiek := CONCAT(sOverKwartierpiek, 's');
ELSE
	sOverKwartierpiek := '';
END_IF

END_PROGRAM

// ---- POUs/08-Energiemetingen/P_Watermeting.TcPOU
PROGRAM P_Watermeting
VAR
	ftWaterSensor		: F_TRIG;
	tonWatermeting		: TON;
	bWatermetingActief	: BOOL;
	rWaterBerekening	: REAL;
END_VAR

ftWaterSensor(CLK:= bWaterSensor , Q=> );

(************************************************************************************************************************)
(************************************************ WATER *************************************************************)
(************************************************************************************************************************)
IF ftWaterSensor.Q THEN
	diWaterteller := diWaterteller + 1;
	(*Stored_Energy[11] := Stored_Energy[11] + 1;	(* Stand watermeter, was vroeger rTotalWaterCounter *)
	rTotalWaterCounter := Stored_Energy[11];*)
END_IF

(* Dagelijks verbruik *)
IF bMiddernacht THEN
	diWatertellerGisteren := diWaterteller;
END_IF
diWaterverbruikVandaag := diWaterteller - diWatertellerGisteren;

(* Liter per uur berekening*)
tonWatermeting(IN:= bWatermetingActief, PT:=t#1m );

IF ftWaterSensor.Q AND tonWatermeting.ET = t#0ms THEN
	bWatermetingActief := TRUE;
ELSIF ftWaterSensor.Q AND bWatermetingActief AND tonWatermeting.ET > t#0ms THEN
	rWaterBerekening := 60000.0 / TIME_TO_UDINT(tonWatermeting.ET);
	(* Berekening waterverbruik per minuut:
										   1Puls = 1Liter
										   1Liter / ElapsedTime(ms) = L/ms * 60000 = L/min            *)

	(* Reset timer voor volgende meting *)
	tonWatermeting(IN:= FALSE );
END_IF

(* Reset na aflopen van de timer, tijd is te lang tussen 2 pulsen *)
IF  tonWatermeting.Q THEN
	bWatermetingActief := FALSE;
	rWaterBerekening := 0;
END_IF

END_PROGRAM

// ---- POUs/09-Ventilatie/P_Ventilatie.TcPOU
PROGRAM P_Ventilatie
VAR
	rVolt			: REAL;
	rtVentUP		: R_TRIG;
	rtVentDOWN		: R_TRIG;

	iVentLOW		: INT := 20;
	iVentHIGH		: INT := 20;
	iVentPrevious	: INT := 20;
	rtLampDouche	: R_TRIG;
	ftLampDouche	: F_TRIG;
	bDouche			: BOOL;
END_VAR

(* Ventilatie instellingen:
	Proportionele ingang 1:
		CO2 meting
		Boost limit: 2000
		Normal limit: 1000
	INT Uitgang:
		9100 = minimale waarde = 20%
		32000 = maximale waarde = 100%					
*)

rtLampDouche(CLK:= bNovRamLight_W5 , Q=> );
ftLampDouche(CLK:= bNovRamLight_W5 , Q=> );

rtVentUP(CLK:= bDK05x4 OR bVentUP, Q=> );
rtVentDOWN(CLK:= bDK05x3 OR bVentDOWN, Q=> );

IF rtLampDouche.Q AND (todWinTime < tod#19:00:00) AND (todWinTime > tod#08:00:00) THEN
	iVentPrevious := iNovRamVentilatie;
	iNovRamVentilatie := 60;
	bDouche := TRUE;
ELSIF ftLampDouche.Q AND bDouche THEN
	iNovRamVentilatie := iVentPrevious;
	bDouche := FALSE;
END_IF

IF todWinTime = tod#19:00 THEN
	iNovRamVentilatie := iVentLOW;
	bDouche := FALSE;
ELSIF todWinTime = tod#10:00 AND (iNovRamVentilatie < iVentHIGH) THEN
	iNovRamVentilatie := iVentHIGH;
END_IF

IF rtVentUP.Q AND iNovRamVentilatie <= 90 THEN
	iNovRamVentilatie := iNovRamVentilatie + 10;
ELSIF rtVentDOWN.Q AND iNovRamVentilatie >= 30 THEN
	iNovRamVentilatie := iNovRamVentilatie - 10;
END_IF

CASE iNovRamVentilatie OF
20:
	iVentilatie := 0;
30:
	iVentilatie := 12000;
40:
	iVentilatie := 15000;
50:
	iVentilatie := 17600;
60:
	iVentilatie := 20500;
70:
	iVentilatie := 23400;
80:
	iVentilatie := 26000;
90:
	iVentilatie := 29000;
100:
	iVentilatie := 32000;
ELSE
	iNovRamVentilatie := 20;
END_CASE

IF iVentilatie < 0 THEN
	iVentilatie := 0;
ELSIF iVentilatie > 32000 THEN
	iVentilatie := 32000;
END_IF

rVolt := INT_TO_REAL(iVentilatie)/3276.7;

END_PROGRAM

// ---- POUs/10-IoT/P_IoT_Communicator.TcPOU
PROGRAM P_IoT_Communicator
VAR
	fbIoT : FB_IotCommunicator := (
		sHostName := 'k3a60711.ala.eu-central-1.emqxsl.com', 	// MQTT Broker Adress
		nPort := 8883,                   						// MQTT Port
		sClientId := 'btn000u5j7t', 
		sMainTopic := 'Beestenboel',          					// Main Topic
		sDeviceName := 'btn000u5j7t',  							// Device Name
		sUser := 'BeckhoffCX7000',            					// MQTT Username
		sPassword := 'N6u57nyWUtum25v');         				// MQTT Password

	stData	: ST_IoT_Communicator;              				// Values to send
	timer 	: TON;                         						// Timer to send data
END_VAR

fbIoT.stTls.bNoServerCertCheck := TRUE;
fbIoT.Execute(TRUE);

timer(IN := NOT timer.Q, PT := T#500MS);

IF fbIoT.bConnected AND timer.Q THEN
    fbIoT.SendData(ADR(stData), SIZEOF(stData));
END_IF

stData.rActiefVermogen := P_Kwartierpiek.CurrentActivePower;

END_PROGRAM
